C03579=1018.745,297.006,-138.306,170.005,50.463,159.764
C03580=1018.752,297.252,-138.337,170.011,50.459,159.764
C03581=1018.758,297.501,-138.369,170.016,50.455,159.763
C03582=1018.764,297.748,-138.401,170.022,50.451,159.763
C03583=1018.770,297.997,-138.433,170.026,50.447,159.763
C03584=1018.777,298.245,-138.464,170.033,50.443,159.764
C03585=1018.783,298.492,-138.497,170.038,50.439,159.764
C03586=1018.789,298.740,-138.529,170.043,50.435,159.764
C03587=1018.795,298.988,-138.560,170.048,50.431,159.763
C03588=1018.801,299.236,-138.592,170.055,50.427,159.764
C03589=1018.808,299.483,-138.624,170.059,50.423,159.764
C03590=1018.814,299.731,-138.656,170.065,50.418,159.764
C03591=1018.821,299.979,-138.688,170.071,50.414,159.764
C03592=1018.827,300.227,-138.720,170.076,50.411,159.764
C03593=1018.833,300.475,-138.753,170.082,50.406,159.764
C03594=1018.840,300.723,-138.784,170.087,50.402,159.764
C03595=1018.846,300.970,-138.817,170.094,50.399,159.764
C03596=1018.853,301.218,-138.848,170.098,50.395,159.764
C03597=1018.859,301.467,-138.880,170.104,50.390,159.764
C03598=1018.866,301.714,-138.912,170.110,50.387,159.764
C03599=1018.872,301.962,-138.944,170.115,50.383,159.764
C03600=1018.879,302.210,-138.977,170.121,50.379,159.764
C03601=1018.885,302.458,-139.009,170.127,50.375,159.764
C03602=1018.892,302.705,-139.041,170.132,50.371,159.764
C03603=1018.898,302.953,-139.073,170.138,50.367,159.764
C03604=1018.905,303.201,-139.105,170.144,50.363,159.764
C03605=1018.911,303.449,-139.137,170.149,50.360,159.764
C03606=1018.918,303.696,-139.170,170.155,50.355,159.764
C03607=1018.924,303.944,-139.202,170.160,50.352,159.764
C03608=1018.931,304.192,-139.234,170.166,50.348,159.764
C03609=1018.937,304.440,-139.266,170.171,50.344,159.764
C03610=1018.944,304.687,-139.298,170.177,50.341,159.765
C03611=1018.950,304.935,-139.331,170.183,50.336,159.765
C03612=1018.957,305.183,-139.363,170.189,50.333,159.765
C03613=1018.964,305.431,-139.395,170.194,50.328,159.765
C03614=1018.970,305.679,-139.428,170.200,50.325,159.765
C03615=1018.977,305.926,-139.459,170.206,50.321,159.765
C03616=1018.983,306.174,-139.492,170.212,50.317,159.765
C03617=1018.990,306.421,-139.524,170.217,50.314,159.765
C03618=1018.997,306.670,-139.557,170.223,50.309,159.765
C03619=1019.003,306.917,-139.589,170.228,50.306,159.765
C03620=1019.010,307.163,-139.621,170.235,50.302,159.765
C03621=1019.016,307.409,-139.653,170.240,50.299,159.766
C03622=1019.023,307.655,-139.686,170.246,50.295,159.765
C03623=1019.030,307.901,-139.718,170.251,50.291,159.766
C03624=1019.036,308.146,-139.751,170.257,50.288,159.766
C03625=1019.043,308.391,-139.783,170.263,50.284,159.766
C03626=1019.050,308.637,-139.815,170.268,50.280,159.766
C03627=1019.057,308.884,-139.847,170.275,50.276,159.766
C03628=1019.063,309.131,-139.880,170.280,50.273,159.766
C03629=1019.070,309.379,-139.912,170.286,50.269,159.766
C03630=1019.076,309.626,-139.944,170.292,50.266,159.767
C03631=1019.083,309.874,-139.977,170.297,50.262,159.767
C03632=1019.090,310.122,-140.011,170.304,50.258,159.767
C03633=1019.096,310.369,-140.044,170.309,50.255,159.767
C03634=1019.102,310.617,-140.076,170.315,50.252,159.767
C03635=1019.109,310.864,-140.110,170.321,50.248,159.767
C03636=1019.115,311.112,-140.144,170.327,50.245,159.768
C03637=1019.121,311.360,-140.176,170.332,50.241,159.768
C03638=1019.128,311.607,-140.210,170.339,50.238,159.768
C03639=1019.135,311.855,-140.243,170.344,50.234,159.768
C03640=1019.141,312.103,-140.276,170.350,50.231,159.768
C03641=1019.147,312.350,-140.310,170.356,50.228,159.768
C03642=1019.154,312.598,-140.343,170.362,50.224,159.769
C03643=1019.161,312.845,-140.376,170.367,50.221,159.769
C03644=1019.167,313.093,-140.409,170.374,50.217,159.769
C03645=1019.173,313.342,-140.443,170.379,50.215,159.769
C03646=1019.180,313.589,-140.476,170.385,50.211,159.769
C03647=1019.186,313.837,-140.509,170.391,50.208,159.770
C03648=1019.193,314.084,-140.543,170.397,50.204,159.770
C03649=1019.200,314.331,-140.576,170.404,50.201,159.770
C03650=1019.206,314.579,-140.610,170.409,50.197,159.770
C03651=1019.212,314.826,-140.643,170.415,50.194,159.770
C03652=1019.219,315.075,-140.677,170.421,50.191,159.771
C03653=1019.226,315.322,-140.710,170.427,50.187,159.771
C03654=1019.232,315.570,-140.744,170.433,50.185,159.771
C03655=1019.239,315.817,-140.777,170.439,50.181,159.771
C03656=1019.246,316.065,-140.811,170.444,50.178,159.772
C03657=1019.252,316.312,-140.844,170.451,50.175,159.772
C03658=1019.259,316.560,-140.878,170.457,50.171,159.772
C03659=1019.265,316.807,-140.912,170.463,50.168,159.772
C03660=1019.272,317.056,-140.945,170.469,50.165,159.773
C03661=1019.279,317.303,-140.979,170.475,50.162,159.773
C03662=1019.285,317.551,-141.013,170.481,50.158,159.773
C03663=1019.292,317.798,-141.046,170.487,50.156,159.773
C03664=1019.299,318.046,-141.079,170.493,50.152,159.774
C03665=1019.306,318.294,-141.113,170.500,50.149,159.774
C03666=1019.312,318.542,-141.147,170.505,50.146,159.774
C03667=1019.319,318.789,-141.181,170.512,50.143,159.775
C03668=1019.326,319.036,-141.215,170.518,50.139,159.775
C03669=1019.333,319.284,-141.248,170.523,50.136,159.775
C03670=1019.339,319.531,-141.283,170.530,50.133,159.775
C03671=1019.346,319.779,-141.316,170.535,50.130,159.776
C03672=1019.353,320.027,-141.349,170.542,50.127,159.776
C03673=1019.360,320.274,-141.383,170.549,50.124,159.776
C03674=1019.366,320.522,-141.417,170.554,50.121,159.776
C03675=1019.374,320.770,-141.451,170.561,50.118,159.777
C03676=1019.381,321.017,-141.485,170.566,50.115,159.777
C03677=1019.387,321.264,-141.518,170.572,50.111,159.777
C03678=1019.394,321.512,-141.553,170.579,50.108,159.778
C03679=1019.401,321.760,-141.587,170.585,50.106,159.778
C03680=1019.408,322.009,-141.621,170.591,50.103,159.778
C03681=1019.415,322.258,-141.656,170.598,50.099,159.779
C03682=1019.422,322.507,-141.689,170.603,50.096,159.779
C03683=1019.429,322.756,-141.724,170.610,50.093,159.779
C03684=1019.437,323.004,-141.758,170.617,50.090,159.780
C03685=1019.443,323.252,-141.792,170.622,50.088,159.780
C03686=1019.450,323.498,-141.826,170.629,50.084,159.780
C03687=1019.457,323.746,-141.859,170.635,50.081,159.781
C03688=1019.463,323.994,-141.894,170.642,50.078,159.781
C03689=1019.471,324.241,-141.928,170.647,50.075,159.781
C03690=1019.478,324.489,-141.962,170.654,50.072,159.782
C03691=1019.485,324.737,-141.996,170.661,50.069,159.782
C03692=1019.492,324.985,-142.030,170.666,50.066,159.782
C03693=1019.499,325.232,-142.065,170.673,50.063,159.783
C03694=1019.506,325.479,-142.099,170.680,50.060,159.783
C03695=1019.514,325.727,-142.133,170.685,50.058,159.783
C03696=1019.520,325.974,-142.168,170.692,50.055,159.784
C03697=1019.528,326.222,-142.202,170.699,50.052,159.784
C03698=1019.535,326.469,-142.236,170.704,50.049,159.784
C03699=1019.542,326.717,-142.270,170.711,50.046,159.785
C03700=1019.548,326.964,-142.306,170.718,50.043,159.785
C03701=1019.555,327.212,-142.339,170.724,50.041,159.786
C03702=1019.562,327.459,-142.375,170.730,50.038,159.786
C03703=1019.569,327.707,-142.410,170.737,50.035,159.787
C03704=1019.576,327.954,-142.444,170.743,50.032,159.787
C03705=1019.583,328.202,-142.479,170.750,50.030,159.787
C03706=1019.590,328.449,-142.514,170.756,50.027,159.788
C03707=1019.597,328.697,-142.549,170.762,50.024,159.788
C03708=1019.604,328.944,-142.583,170.769,50.022,159.789
C03709=1019.610,329.192,-142.618,170.776,50.019,159.789
C03710=1019.617,329.439,-142.653,170.781,50.016,159.789
C03711=1019.625,329.686,-142.688,170.788,50.014,159.790
C03712=1019.632,329.933,-142.723,170.795,50.011,159.790
C03713=1019.639,330.182,-142.758,170.801,50.009,159.791
C03714=1019.645,330.429,-142.793,170.808,50.006,159.791
C03715=1019.653,330.676,-142.827,170.814,50.003,159.792
C03716=1019.660,330.924,-142.862,170.821,50.000,159.792
C03717=1019.666,331.171,-142.897,170.827,49.998,159.793
C03718=1019.673,331.419,-142.933,170.834,49.995,159.793
C03719=1019.681,331.666,-142.967,170.841,49.992,159.793
C03720=1019.688,331.914,-143.003,170.847,49.990,159.794
C03721=1019.695,332.161,-143.038,170.853,49.987,159.794
C03722=1019.702,332.408,-143.072,170.860,49.985,159.795
C03723=1019.710,332.656,-143.108,170.867,49.983,159.796
C03724=1019.716,332.904,-143.143,170.873,49.980,159.796
C03725=1019.723,333.151,-143.178,170.880,49.978,159.796
C03726=1019.730,333.398,-143.214,170.887,49.975,159.797
C03727=1019.738,333.646,-143.249,170.893,49.972,159.797
C03728=1019.744,333.893,-143.285,170.900,49.970,159.798
C03729=1019.751,334.140,-143.320,170.907,49.968,159.798
C03730=1019.758,334.387,-143.356,170.914,49.965,159.799
C03731=1019.766,334.635,-143.391,170.919,49.963,159.799
C03732=1019.772,334.883,-143.426,170.926,49.960,159.800
C03733=1019.779,335.129,-143.462,170.933,49.958,159.801
C03734=1019.787,335.377,-143.498,170.939,49.956,159.801
C03735=1019.794,335.625,-143.533,170.946,49.954,159.802
C03736=1019.801,335.872,-143.569,170.953,49.951,159.802
C03737=1019.808,336.120,-143.604,170.960,49.948,159.803
C03738=1019.815,336.366,-143.640,170.966,49.946,159.803
C03739=1019.823,336.614,-143.675,170.973,49.944,159.804
C03740=1019.830,336.860,-143.710,170.980,49.941,159.804
C03741=1019.837,337.106,-143.747,170.987,49.939,159.805
C03742=1019.844,337.352,-143.782,170.993,49.937,159.805
C03743=1019.851,337.599,-143.818,171.000,49.935,159.806
C03744=1019.859,337.844,-143.852,171.007,49.932,159.806
C03745=1019.866,338.091,-143.888,171.014,49.930,159.807
C03746=1019.873,338.336,-143.924,171.020,49.928,159.808
C03747=1019.880,338.583,-143.960,171.027,49.926,159.808
C03748=1019.887,338.830,-143.996,171.034,49.923,159.809
C03749=1019.895,339.078,-144.031,171.042,49.921,159.810
C03750=1019.902,339.324,-144.067,171.049,49.919,159.810
C03751=1019.909,339.572,-144.103,171.055,49.917,159.811
C03752=1019.917,339.819,-144.139,171.062,49.915,159.811
C03753=1019.924,340.066,-144.176,171.069,49.912,159.812
C03754=1019.931,340.315,-144.211,171.076,49.911,159.813
C03755=1019.938,340.561,-144.247,171.083,49.908,159.813
C03756=1019.946,340.809,-144.283,171.089,49.906,159.814
C03757=1019.952,341.056,-144.320,171.096,49.904,159.814
C03758=1019.960,341.303,-144.356,171.104,49.902,159.815
C03759=1019.967,341.551,-144.392,171.111,49.900,159.816
C03760=1019.974,341.797,-144.428,171.118,49.897,159.816
C03761=1019.981,342.045,-144.465,171.124,49.896,159.817
C03762=1019.989,342.293,-144.501,171.131,49.894,159.817
C03763=1019.996,342.539,-144.537,171.139,49.892,159.818
C03764=1020.004,342.786,-144.574,171.146,49.889,159.819
C03765=1020.011,343.034,-144.611,171.153,49.888,159.820
C03766=1020.018,343.281,-144.647,171.160,49.885,159.820
C03767=1020.026,343.528,-144.683,171.166,49.884,159.821
C03768=1020.033,343.776,-144.720,171.173,49.882,159.821
C03769=1020.040,344.023,-144.756,171.181,49.880,159.822
C03770=1020.048,344.269,-144.792,171.188,49.877,159.823
C03771=1020.055,344.517,-144.829,171.195,49.876,159.824
C03772=1020.062,344.765,-144.865,171.202,49.873,159.824
C03773=1020.070,345.011,-144.902,171.210,49.872,159.825
C03774=1020.077,345.259,-144.939,171.217,49.870,159.826
C03775=1020.085,345.507,-144.975,171.223,49.868,159.826
C03776=1020.092,345.753,-145.012,171.230,49.866,159.827
C03777=1020.099,346.001,-145.049,171.238,49.864,159.828
C03778=1020.107,346.247,-145.086,171.245,49.862,159.828
C03779=1020.115,346.495,-145.122,171.252,49.860,159.829
C03780=1020.122,346.742,-145.159,171.260,49.859,159.830
C03781=1020.130,346.989,-145.196,171.267,49.857,159.831
C03782=1020.138,347.236,-145.233,171.274,49.854,159.831
C03783=1020.145,347.484,-145.269,171.281,49.853,159.832
C03784=1020.152,347.731,-145.307,171.289,49.851,159.833
C03785=1020.160,347.978,-145.344,171.296,49.849,159.834
C03786=1020.167,348.226,-145.381,171.304,49.848,159.834
C03787=1020.175,348.473,-145.418,171.310,49.846,159.835
C03788=1020.182,348.720,-145.455,171.317,49.844,159.836
C03789=1020.190,348.966,-145.492,171.325,49.843,159.837
C03790=1020.197,349.214,-145.529,171.332,49.841,159.837
C03791=1020.205,349.461,-145.566,171.340,49.839,159.838
C03792=1020.212,349.708,-145.603,171.347,49.837,159.839
C03793=1020.220,349.955,-145.641,171.354,49.836,159.840
C03794=1020.228,350.202,-145.678,171.362,49.834,159.841
C03795=1020.235,350.449,-145.715,171.369,49.832,159.841
C03796=1020.242,350.696,-145.753,171.376,49.830,159.842
C03797=1020.250,350.943,-145.790,171.384,49.829,159.843
C03798=1020.257,351.190,-145.827,171.392,49.828,159.844
C03799=1020.265,351.437,-145.864,171.399,49.826,159.845
C03800=1020.272,351.682,-145.901,171.406,49.824,159.845
C03801=1020.280,351.927,-145.938,171.414,49.822,159.846
C03802=1020.288,352.171,-145.975,171.421,49.821,159.847
C03803=1020.295,352.416,-146.012,171.429,49.820,159.848
C03804=1020.302,352.661,-146.049,171.436,49.818,159.849
C03805=1020.310,352.905,-146.086,171.444,49.816,159.850
C03806=1020.318,353.150,-146.124,171.451,49.814,159.850
C03807=1020.326,353.394,-146.161,171.459,49.813,159.851
C03808=1020.334,353.641,-146.198,171.466,49.811,159.852
C03809=1020.341,353.888,-146.236,171.474,49.810,159.853
C03810=1020.350,354.135,-146.274,171.481,49.809,159.854
C03811=1020.357,354.382,-146.311,171.489,49.807,159.855
C03812=1020.364,354.629,-146.349,171.497,49.806,159.856
C03813=1020.372,354.876,-146.387,171.504,49.804,159.856
C03814=1020.380,355.124,-146.425,171.512,49.803,159.857
C03815=1020.388,355.370,-146.463,171.519,49.801,159.858
C03816=1020.395,355.617,-146.500,171.527,49.800,159.859
C03817=1020.403,355.864,-146.539,171.535,49.799,159.860
C03818=1020.410,356.111,-146.576,171.542,49.797,159.861
C03819=1020.418,356.358,-146.614,171.550,49.796,159.862
C03820=1020.427,356.605,-146.652,171.557,49.794,159.863
C03821=1020.434,356.852,-146.690,171.566,49.793,159.864
C03822=1020.442,357.099,-146.729,171.574,49.792,159.865
C03823=1020.450,357.346,-146.766,171.582,49.791,159.866
C03824=1020.458,357.594,-146.805,171.589,49.789,159.866
C03825=1020.465,357.840,-146.843,171.597,49.788,159.867
C03826=1020.474,358.087,-146.881,171.604,49.787,159.868
C03827=1020.481,358.334,-146.919,171.612,49.785,159.869
C03828=1020.490,358.581,-146.957,171.620,49.784,159.870
C03829=1020.497,358.828,-146.995,171.628,49.782,159.871
C03830=1020.505,359.075,-147.034,171.636,49.781,159.872
C03831=1020.513,359.322,-147.072,171.644,49.780,159.873
C03832=1020.521,359.569,-147.111,171.652,49.779,159.874
C03833=1020.529,359.815,-147.149,171.659,49.778,159.875
C03834=1020.537,360.063,-147.188,171.667,49.777,159.876
C03835=1020.544,360.309,-147.226,171.676,49.775,159.877
C03836=1020.552,360.556,-147.265,171.684,49.774,159.878
C03837=1020.561,360.803,-147.303,171.691,49.773,159.879
C03838=1020.568,361.050,-147.341,171.699,49.772,159.880
C03839=1020.575,361.298,-147.381,171.707,49.771,159.881
C03840=1020.583,361.543,-147.420,171.716,49.770,159.882
C03841=1020.591,361.791,-147.458,171.724,49.769,159.883
C03842=1020.600,362.038,-147.497,171.732,49.768,159.884
C03843=1020.607,362.284,-147.535,171.739,49.766,159.885
C03844=1020.616,362.531,-147.574,171.747,49.765,159.886
C03845=1020.624,362.778,-147.613,171.756,49.764,159.888
C03846=1020.631,363.025,-147.651,171.764,49.763,159.889
C03847=1020.639,363.272,-147.691,171.772,49.762,159.890
C03848=1020.647,363.519,-147.730,171.780,49.762,159.891
C03849=1020.656,363.765,-147.769,171.789,49.760,159.892
C03850=1020.664,364.013,-147.808,171.796,49.759,159.893
C03851=1020.672,364.258,-147.847,171.805,49.759,159.894
C03852=1020.680,364.506,-147.885,171.813,49.757,159.895
C03853=1020.688,364.752,-147.925,171.821,49.757,159.896
C03854=1020.696,365.000,-147.964,171.829,49.755,159.897
C03855=1020.704,365.246,-148.003,171.837,49.754,159.898
C03856=1020.713,365.493,-148.042,171.846,49.753,159.899
C03857=1020.721,365.740,-148.081,171.854,49.752,159.900
C03858=1020.729,365.986,-148.120,171.862,49.752,159.902
C03859=1020.737,366.233,-148.159,171.871,49.751,159.903
C03860=1020.745,366.482,-148.199,171.879,49.750,159.904
C03861=1020.753,366.732,-148.238,171.888,49.749,159.905
C03862=1020.762,366.981,-148.278,171.896,49.748,159.906
C03863=1020.770,367.231,-148.318,171.905,49.747,159.907
C03864=1020.779,367.478,-148.357,171.913,49.746,159.908
C03865=1020.787,367.725,-148.397,171.921,49.746,159.910
C03866=1020.796,367.971,-148.436,171.930,49.744,159.911
C03867=1020.804,368.218,-148.476,171.938,49.744,159.912
C03868=1020.812,368.465,-148.515,171.947,49.743,159.913
C03869=1020.820,368.712,-148.555,171.955,49.742,159.914
C03870=1020.828,368.958,-148.594,171.963,49.742,159.916
C03871=1020.836,369.205,-148.634,171.973,49.741,159.917
C03872=1020.845,369.451,-148.674,171.981,49.741,159.918
C03873=1020.852,369.698,-148.714,171.990,49.740,159.919
C03874=1020.861,369.945,-148.754,171.998,49.739,159.920
C03875=1020.869,370.192,-148.793,172.007,49.738,159.922
C03876=1020.877,370.437,-148.833,172.015,49.738,159.923
C03877=1020.885,370.684,-148.873,172.023,49.737,159.924
C03878=1020.894,370.932,-148.913,172.033,49.736,159.925
C03879=1020.902,371.178,-148.954,172.041,49.736,159.927
C03880=1020.911,371.425,-148.993,172.050,49.735,159.928
C03881=1020.919,371.671,-149.034,172.058,49.734,159.929
C03882=1020.927,371.917,-149.073,172.067,49.734,159.930
C03883=1020.936,372.165,-149.113,172.076,49.734,159.932
C03884=1020.944,372.411,-149.153,172.085,49.733,159.933
C03885=1020.953,372.657,-149.193,172.093,49.732,159.934
C03886=1020.961,372.905,-149.234,172.102,49.732,159.936
C03887=1020.970,373.151,-149.274,172.111,49.731,159.937
C03888=1020.978,373.397,-149.314,172.120,49.731,159.938
C03889=1020.987,373.644,-149.354,172.129,49.730,159.939
C03890=1020.995,373.890,-149.395,172.137,49.730,159.941
C03891=1021.004,374.137,-149.434,172.146,49.729,159.942
C03892=1021.012,374.384,-149.475,172.155,49.729,159.943
C03893=1021.021,374.630,-149.515,172.164,49.728,159.945
C03894=1021.030,374.877,-149.556,172.173,49.728,159.946
C03895=1021.038,375.123,-149.596,172.182,49.727,159.947
C03896=1021.047,375.371,-149.636,172.191,49.727,159.949
C03897=1021.055,375.617,-149.676,172.200,49.726,159.950
C03898=1021.064,375.864,-149.717,172.209,49.726,159.951
C03899=1021.073,376.110,-149.757,172.218,49.725,159.953
C03900=1021.081,376.357,-149.798,172.227,49.725,159.954
C03901=1021.089,376.603,-149.839,172.236,49.725,159.955
C03902=1021.098,376.850,-149.880,172.245,49.725,159.957
C03903=1021.107,377.095,-149.921,172.254,49.724,159.958
C03904=1021.116,377.342,-149.962,172.263,49.724,159.960
C03905=1021.124,377.588,-150.002,172.272,49.724,159.961
C03906=1021.132,377.835,-150.043,172.282,49.723,159.962
C03907=1021.141,378.081,-150.085,172.290,49.723,159.964
C03908=1021.150,378.328,-150.125,172.300,49.723,159.965
C03909=1021.159,378.575,-150.166,172.309,49.723,159.967
C03910=1021.167,378.820,-150.208,172.319,49.723,159.968
C03911=1021.176,379.067,-150.249,172.327,49.723,159.970
C03912=1021.185,379.314,-150.290,172.337,49.722,159.971
C03913=1021.193,379.560,-150.331,172.346,49.722,159.973
C03914=1021.202,379.806,-150.372,172.356,49.722,159.974
C03915=1021.211,380.053,-150.413,172.364,49.722,159.975
C03916=1021.219,380.299,-150.454,172.374,49.722,159.977
C03917=1021.228,380.545,-150.496,172.383,49.721,159.978
C03918=1021.237,380.792,-150.537,172.393,49.721,159.980
C03919=1021.246,381.038,-150.579,172.403,49.721,159.982
C03920=1021.256,381.310,-150.624,172.412,49.721,159.983
C03921=1021.265,381.581,-150.669,172.423,49.721,159.985
C03922=1021.276,381.852,-150.715,172.434,49.721,159.986
C03923=1021.285,382.124,-150.761,172.444,49.721,159.988
C03924=1021.294,382.370,-150.803,172.453,49.721,159.990
C03925=1021.303,382.617,-150.844,172.463,49.721,159.991
C03926=1021.313,382.863,-150.885,172.473,49.721,159.993
C03927=1021.322,383.109,-150.927,172.482,49.721,159.994
C03928=1021.331,383.356,-150.969,172.492,49.720,159.996
C03929=1021.339,383.602,-151.010,172.502,49.721,159.997
C03930=1021.348,383.848,-151.052,172.511,49.720,159.999
C03931=1021.357,384.095,-151.094,172.521,49.721,160.001
C03932=1021.367,384.341,-151.135,172.531,49.721,160.002
C03933=1021.376,384.587,-151.177,172.540,49.721,160.004
C03934=1021.385,384.833,-151.218,172.550,49.721,160.005
C03935=1021.394,385.080,-151.260,172.560,49.721,160.007
C03936=1021.403,385.326,-151.302,172.570,49.721,160.008
C03937=1021.412,385.573,-151.344,172.580,49.721,160.010
C03938=1021.421,385.819,-151.386,172.589,49.721,160.012
C03939=1021.430,386.065,-151.428,172.599,49.721,160.013
C03940=1021.440,386.311,-151.471,172.609,49.721,160.015
C03941=1021.449,386.558,-151.512,172.619,49.722,160.017
C03942=1021.458,386.803,-151.555,172.629,49.722,160.018
C03943=1021.467,387.050,-151.597,172.638,49.722,160.020
C03944=1021.477,387.296,-151.639,172.648,49.723,160.022
C03945=1021.486,387.542,-151.681,172.658,49.723,160.023
C03946=1021.495,387.788,-151.723,172.669,49.723,160.025
C03947=1021.505,388.035,-151.766,172.679,49.723,160.027
C03948=1021.513,388.281,-151.808,172.689,49.723,160.028
C03949=1021.522,388.527,-151.851,172.699,49.724,160.030
C03950=1021.531,388.773,-151.893,172.709,49.724,160.032
C03951=1021.541,389.019,-151.936,172.719,49.725,160.034
C03952=1021.550,389.265,-151.979,172.729,49.725,160.035
C03953=1021.559,389.512,-152.022,172.740,49.725,160.037
C03954=1021.569,389.757,-152.064,172.749,49.725,160.039
C03955=1021.578,390.003,-152.107,172.760,49.726,160.041
C03956=1021.588,390.250,-152.150,172.770,49.726,160.042
C03957=1021.596,390.496,-152.193,172.781,49.727,160.044
C03958=1021.606,390.742,-152.235,172.791,49.727,160.046
C03959=1021.615,390.988,-152.278,172.801,49.727,160.048
C03960=1021.625,391.234,-152.321,172.811,49.728,160.050
C03961=1021.634,391.480,-152.363,172.822,49.728,160.051
C03962=1021.644,391.727,-152.407,172.832,49.729,160.053
C03963=1021.653,391.972,-152.450,172.842,49.730,160.055
C03964=1021.663,392.218,-152.492,172.853,49.730,160.057
C03965=1021.671,392.464,-152.536,172.863,49.731,160.059
C03966=1021.682,392.710,-152.579,172.873,49.731,160.060
C03967=1021.691,392.957,-152.622,172.884,49.732,160.062
C03968=1021.700,393.202,-152.666,172.895,49.732,160.064
C03969=1021.710,393.449,-152.708,172.905,49.733,160.066
C03970=1021.720,393.694,-152.752,172.916,49.734,160.068
C03971=1021.729,393.940,-152.795,172.926,49.734,160.070
C03972=1021.739,394.186,-152.838,172.937,49.734,160.072
C03973=1021.748,394.432,-152.883,172.948,49.735,160.074
C03974=1021.758,394.679,-152.925,172.958,49.736,160.076
C03975=1021.767,394.924,-152.969,172.969,49.737,160.078
C03976=1021.777,395.170,-153.013,172.979,49.737,160.079
C03977=1021.787,395.416,-153.056,172.990,49.738,160.081
C03978=1021.796,395.663,-153.099,173.001,49.739,160.083
C03979=1021.806,395.909,-153.143,173.012,49.739,160.085
C03980=1021.819,396.217,-153.198,173.026,49.740,160.088
C03981=1021.831,396.525,-153.253,173.039,49.742,160.090
C03982=1021.843,396.834,-153.307,173.053,49.743,160.093
C03983=1021.855,397.142,-153.363,173.067,49.744,160.095
C03984=1021.865,397.388,-153.407,173.078,49.744,160.097
C03985=1021.875,397.634,-153.450,173.088,49.745,160.099
C03986=1021.884,397.880,-153.494,173.100,49.746,160.101
C03987=1021.895,398.126,-153.539,173.110,49.747,160.103
C03988=1021.904,398.372,-153.583,173.122,49.748,160.105
C03989=1021.914,398.618,-153.627,173.133,49.748,160.107
C03990=1021.924,398.863,-153.671,173.144,49.750,160.110
C03991=1021.934,399.109,-153.715,173.155,49.750,160.111
C03992=1021.944,399.355,-153.759,173.167,49.751,160.114
C03993=1021.954,399.601,-153.804,173.177,49.752,160.116
C03994=1021.964,399.847,-153.849,173.189,49.753,160.118
C03995=1021.974,400.093,-153.892,173.200,49.754,160.120
C03996=1021.984,400.338,-153.937,173.212,49.755,160.122
C03997=1021.993,400.584,-153.981,173.222,49.756,160.124
C03998=1022.004,400.830,-154.026,173.234,49.757,160.126
C03999=1022.014,401.076,-154.071,173.245,49.758,160.128
C04000=1022.024,401.321,-154.115,173.257,49.759,160.131
C04001=1022.033,401.567,-154.160,173.269,49.760,160.133
C04002=1022.043,401.814,-154.205,173.279,49.762,160.135
C04003=1022.053,402.059,-154.249,173.291,49.763,160.137
C04004=1022.063,402.304,-154.294,173.302,49.764,160.139
C04005=1022.074,402.550,-154.339,173.314,49.765,160.141
C04006=1022.084,402.795,-154.384,173.326,49.766,160.144
C04007=1022.093,403.041,-154.429,173.338,49.767,160.146
C04008=1022.104,403.287,-154.474,173.349,49.768,160.148
C04009=1022.114,403.532,-154.519,173.361,49.769,160.150
C04010=1022.125,403.778,-154.564,173.373,49.770,160.152
C04011=1022.134,404.024,-154.609,173.385,49.772,160.155
C04012=1022.145,404.270,-154.655,173.396,49.773,160.157
C04013=1022.155,404.515,-154.699,173.408,49.774,160.159
C04014=1022.165,404.761,-154.745,173.420,49.776,160.162
C04015=1022.176,405.006,-154.790,173.431,49.777,160.164
C04016=1022.186,405.252,-154.835,173.443,49.778,160.166
C04017=1022.196,405.497,-154.880,173.455,49.779,160.168
C04018=1022.206,405.743,-154.925,173.467,49.781,160.171
C04019=1022.217,405.989,-154.971,173.479,49.782,160.173
C04020=1022.227,406.235,-155.017,173.491,49.783,160.175
C04021=1022.237,406.480,-155.062,173.503,49.785,160.178
C04022=1022.249,406.725,-155.107,173.516,49.786,160.180
C04023=1022.259,406.971,-155.153,173.527,49.787,160.182
C04024=1022.270,407.217,-155.199,173.539,49.789,160.185
C04025=1022.280,407.462,-155.244,173.551,49.790,160.187
C04026=1022.290,407.708,-155.290,173.563,49.792,160.190
C04027=1022.301,407.954,-155.335,173.576,49.793,160.192
C04028=1022.312,408.199,-155.380,173.588,49.795,160.194
C04029=1022.323,408.445,-155.426,173.600,49.796,160.197
C04030=1022.333,408.690,-155.472,173.613,49.798,160.199
C04031=1022.344,408.936,-155.518,173.625,49.799,160.202
C04032=1022.354,409.181,-155.564,173.637,49.801,160.204
C04033=1022.365,409.427,-155.610,173.650,49.802,160.207
C04034=1022.376,409.672,-155.657,173.662,49.803,160.209
C04035=1022.387,409.918,-155.703,173.675,49.806,160.212
C04036=1022.397,410.163,-155.748,173.688,49.807,160.214
C04037=1022.407,410.408,-155.796,173.700,49.808,160.216
C04038=1022.418,410.654,-155.842,173.712,49.811,160.219
C04039=1022.429,410.899,-155.888,173.725,49.812,160.222
C04040=1022.444,411.231,-155.951,173.743,49.814,160.225
C04041=1022.458,411.561,-156.013,173.760,49.816,160.228
C04042=1022.473,411.893,-156.076,173.776,49.819,160.232
C04043=1022.488,412.224,-156.139,173.794,49.821,160.235
C04044=1022.498,412.470,-156.186,173.807,49.823,160.238
C04045=1022.509,412.715,-156.232,173.819,49.825,160.241
C04046=1022.520,412.960,-156.279,173.833,49.826,160.243
C04047=1022.531,413.206,-156.326,173.846,49.828,160.246
C04048=1022.542,413.451,-156.372,173.858,49.830,160.248
C04049=1022.554,413.697,-156.419,173.871,49.831,160.251
C04050=1022.564,413.942,-156.467,173.885,49.833,160.254
C04051=1022.575,414.187,-156.513,173.897,49.835,160.256
C04052=1022.587,414.433,-156.560,173.911,49.837,160.259
C04053=1022.598,414.678,-156.607,173.924,49.839,160.262
C04054=1022.609,414.923,-156.654,173.937,49.840,160.264
C04055=1022.621,415.169,-156.701,173.950,49.842,160.267
C04056=1022.631,415.414,-156.748,173.964,49.845,160.270
C04057=1022.643,415.659,-156.796,173.977,49.847,160.273
C04058=1022.653,415.905,-156.843,173.990,49.848,160.275
C04059=1022.665,416.150,-156.891,174.004,49.851,160.278
C04060=1022.676,416.395,-156.938,174.017,49.852,160.281
C04061=1022.687,416.640,-156.986,174.031,49.855,160.284
C04062=1022.698,416.886,-157.033,174.044,49.857,160.286
C04063=1022.709,417.131,-157.081,174.057,49.859,160.289
C04064=1022.721,417.375,-157.128,174.071,49.861,160.292
C04065=1022.731,417.621,-157.176,174.085,49.863,160.295
C04066=1022.743,417.866,-157.224,174.098,49.865,160.298
C04067=1022.755,418.111,-157.271,174.112,49.867,160.301
C04068=1022.766,418.357,-157.320,174.126,49.869,160.304
C04069=1022.778,418.602,-157.367,174.140,49.871,160.306
C04070=1022.788,418.847,-157.415,174.154,49.873,160.309
C04071=1022.800,419.092,-157.463,174.168,49.875,160.312
C04072=1022.811,419.337,-157.511,174.182,49.878,160.315
C04073=1022.823,419.582,-157.559,174.195,49.880,160.318
C04074=1022.835,419.827,-157.607,174.209,49.882,160.321
C04075=1022.846,420.072,-157.655,174.224,49.884,160.324
C04076=1022.858,420.317,-157.703,174.238,49.886,160.327
C04077=1022.870,420.563,-157.752,174.251,49.888,160.330
C04078=1022.882,420.808,-157.800,174.265,49.891,160.333
C04079=1022.894,421.053,-157.847,174.280,49.893,160.336
C04080=1022.905,421.298,-157.896,174.294,49.895,160.339
C04081=1022.917,421.543,-157.944,174.308,49.898,160.342
C04082=1022.929,421.789,-157.993,174.323,49.900,160.345
C04083=1022.940,422.034,-158.042,174.337,49.902,160.348
C04084=1022.952,422.278,-158.090,174.352,49.905,160.351
C04085=1022.964,422.523,-158.139,174.366,49.907,160.354
C04086=1022.975,422.769,-158.188,174.380,49.910,160.357
C04087=1022.987,423.013,-158.236,174.395,49.912,160.360
C04088=1022.999,423.258,-158.285,174.409,49.915,160.364
C04089=1023.011,423.503,-158.335,174.424,49.917,160.367
C04090=1023.023,423.748,-158.383,174.439,49.919,160.370
C04091=1023.034,423.993,-158.432,174.453,49.922,160.373
C04092=1023.047,424.238,-158.481,174.469,49.924,160.376
C04093=1023.059,424.483,-158.530,174.483,49.927,160.379
C04094=1023.071,424.728,-158.579,174.498,49.929,160.382
C04095=1023.083,424.972,-158.628,174.513,49.932,160.386
C04096=1023.095,425.217,-158.678,174.528,49.935,160.389
C04097=1023.107,425.463,-158.727,174.543,49.937,160.392
C04098=1023.120,425.708,-158.776,174.558,49.940,160.395
C04099=1023.131,425.952,-158.826,174.573,49.942,160.399
C04100=1023.145,426.222,-158.880,174.590,49.945,160.402
C04101=1023.158,426.491,-158.935,174.607,49.948,160.406
C04102=1023.171,426.761,-158.990,174.623,49.951,160.410
C04103=1023.185,427.031,-159.044,174.640,49.954,160.413
C04104=1023.197,427.275,-159.094,174.655,49.957,160.417
C04105=1023.209,427.520,-159.144,174.670,49.960,160.420
C04106=1023.221,427.764,-159.194,174.686,49.963,160.423
C04107=1023.234,428.009,-159.244,174.701,49.965,160.427
C04108=1023.246,428.254,-159.294,174.717,49.968,160.430
C04109=1023.258,428.499,-159.344,174.732,49.971,160.434
C04110=1023.271,428.744,-159.395,174.749,49.974,160.437
C04111=1023.284,428.988,-159.444,174.764,49.977,160.441
C04112=1023.296,429.233,-159.494,174.780,49.979,160.444
C04113=1023.308,429.478,-159.544,174.796,49.982,160.447
C04114=1023.321,429.722,-159.595,174.811,49.985,160.451
C04115=1023.333,429.967,-159.645,174.827,49.988,160.454
C04116=1023.346,430.212,-159.695,174.843,49.990,160.458
C04117=1023.358,430.456,-159.746,174.859,49.994,160.461
C04118=1023.371,430.700,-159.796,174.875,49.997,160.465
C04119=1023.384,430.945,-159.846,174.892,50.000,160.469
C04120=1023.397,431.190,-159.897,174.907,50.003,160.472
C04121=1023.409,431.434,-159.948,174.924,50.006,160.476
C04122=1023.422,431.678,-159.998,174.940,50.008,160.479
C04123=1023.434,431.923,-160.049,174.956,50.012,160.483
C04124=1023.448,432.168,-160.099,174.973,50.015,160.487
C04125=1023.461,432.413,-160.150,174.989,50.017,160.490
C04126=1023.474,432.657,-160.201,175.005,50.021,160.494
C04127=1023.487,432.901,-160.252,175.022,50.024,160.497
C04128=1023.500,433.146,-160.303,175.038,50.027,160.501
C04129=1023.513,433.390,-160.354,175.055,50.030,160.505
C04130=1023.525,433.636,-160.406,175.072,50.033,160.509
C04131=1023.538,433.879,-160.457,175.088,50.036,160.512
C04132=1023.551,434.124,-160.508,175.105,50.040,160.516
C04133=1023.564,434.369,-160.560,175.122,50.043,160.520
C04134=1023.577,434.612,-160.611,175.139,50.046,160.524
C04135=1023.591,434.857,-160.662,175.156,50.049,160.528
C04136=1023.603,435.101,-160.714,175.172,50.053,160.531
C04137=1023.617,435.345,-160.766,175.190,50.056,160.535
C04138=1023.630,435.590,-160.817,175.206,50.059,160.539
C04139=1023.644,435.834,-160.869,175.224,50.062,160.543
C04140=1023.660,436.152,-160.936,175.247,50.067,160.548
C04141=1023.678,436.468,-161.003,175.269,50.071,160.553
C04142=1023.695,436.786,-161.071,175.291,50.076,160.558
C04143=1023.713,437.103,-161.138,175.314,50.080,160.563
C04144=1023.726,437.347,-161.190,175.332,50.083,160.567
C04145=1023.740,437.592,-161.242,175.349,50.087,160.571
C04146=1023.753,437.836,-161.294,175.366,50.090,160.575
C04147=1023.766,438.080,-161.347,175.384,50.093,160.579
C04148=1023.780,438.324,-161.399,175.402,50.097,160.584
C04149=1023.794,438.568,-161.452,175.420,50.101,160.587
C04150=1023.807,438.812,-161.504,175.438,50.104,160.592
C04151=1023.820,439.056,-161.557,175.456,50.108,160.596
C04152=1023.834,439.301,-161.609,175.474,50.111,160.600
C04153=1023.848,439.545,-161.662,175.492,50.115,160.604
C04154=1023.862,439.788,-161.714,175.510,50.118,160.608
C04155=1023.875,440.032,-161.768,175.528,50.122,160.612
C04156=1023.889,440.277,-161.820,175.547,50.126,160.617
C04157=1023.903,440.521,-161.872,175.565,50.130,160.621
C04158=1023.918,440.765,-161.925,175.583,50.133,160.625
C04159=1023.931,441.009,-161.978,175.602,50.137,160.629
C04160=1023.946,441.268,-162.034,175.621,50.141,160.634
C04161=1023.961,441.529,-162.091,175.641,50.144,160.638
C04162=1023.976,441.789,-162.148,175.661,50.148,160.643
C04163=1023.991,442.047,-162.205,175.680,50.152,160.647
C04164=1023.596,440.124,-162.120,175.526,50.187,160.632
C04165=1023.583,439.880,-162.067,175.508,50.184,160.628
C04166=1023.569,439.636,-162.014,175.490,50.180,160.624
C04167=1023.555,439.391,-161.962,175.472,50.177,160.620
C04168=1023.541,439.147,-161.909,175.453,50.174,160.615
C04169=1023.528,438.903,-161.856,175.436,50.170,160.611
C04170=1023.514,438.659,-161.804,175.417,50.167,160.607
C04171=1023.501,438.415,-161.752,175.400,50.163,160.603
C04172=1023.487,438.171,-161.700,175.382,50.160,160.599
C04173=1023.474,437.927,-161.647,175.364,50.157,160.595
C04174=1023.460,437.682,-161.594,175.347,50.154,160.591
C04175=1023.446,437.438,-161.542,175.329,50.150,160.587
C04176=1023.433,437.194,-161.491,175.311,50.147,160.583
C04177=1023.419,436.949,-161.439,175.294,50.144,160.579
C04178=1023.406,436.705,-161.387,175.276,50.140,160.575
C04179=1023.393,436.461,-161.335,175.259,50.137,160.571
C04180=1023.379,436.217,-161.283,175.242,50.133,160.567
C04181=1023.366,435.973,-161.231,175.225,50.130,160.564
C04182=1023.353,435.728,-161.180,175.207,50.127,160.560
C04183=1023.340,435.483,-161.128,175.190,50.124,160.556
C04184=1023.327,435.240,-161.076,175.173,50.121,160.552
C04185=1023.314,434.995,-161.025,175.156,50.118,160.548
C04186=1023.300,434.751,-160.973,175.139,50.115,160.544
C04187=1023.287,434.506,-160.922,175.122,50.111,160.540
C04188=1023.274,434.262,-160.871,175.105,50.108,160.537
C04189=1023.261,434.017,-160.819,175.088,50.105,160.533
C04190=1023.248,433.773,-160.769,175.071,50.102,160.529
C04191=1023.235,433.529,-160.717,175.055,50.099,160.525
C04192=1023.222,433.285,-160.666,175.038,50.096,160.522
C04193=1023.209,433.040,-160.615,175.021,50.093,160.518
C04194=1023.197,432.795,-160.563,175.005,50.090,160.514
C04195=1023.184,432.551,-160.512,174.988,50.087,160.511
C04196=1023.170,432.306,-160.462,174.972,50.084,160.507
C04197=1023.158,432.062,-160.411,174.956,50.081,160.503
C04198=1023.144,431.817,-160.360,174.939,50.078,160.500
C04199=1023.132,431.572,-160.310,174.923,50.075,160.496
C04200=1023.119,431.328,-160.259,174.906,50.072,160.492
C04201=1023.106,431.083,-160.208,174.891,50.069,160.489
C04202=1023.093,430.839,-160.158,174.874,50.067,160.485
C04203=1023.081,430.595,-160.107,174.858,50.064,160.482
C04204=1023.068,430.350,-160.057,174.841,50.061,160.478
C04205=1023.054,430.093,-160.005,174.825,50.058,160.475
C04206=1023.042,429.838,-159.952,174.809,50.055,160.471
C04207=1023.028,429.583,-159.899,174.792,50.052,160.467
C04208=1023.015,429.327,-159.847,174.775,50.050,160.464
C04209=1023.003,429.082,-159.797,174.760,50.047,160.460
C04210=1022.991,428.837,-159.747,174.744,50.044,160.457
C04211=1022.978,428.592,-159.697,174.728,50.041,160.453
C04212=1022.966,428.348,-159.647,174.712,50.039,160.450
C04213=1022.954,428.103,-159.596,174.697,50.036,160.447
C04214=1022.941,427.858,-159.546,174.681,50.033,160.443
C04215=1022.928,427.613,-159.497,174.666,50.031,160.440
C04216=1022.916,427.369,-159.447,174.650,50.028,160.436
C04217=1022.900,427.040,-159.380,174.630,50.025,160.432
C04218=1022.884,426.711,-159.313,174.609,50.020,160.427
C04219=1022.867,426.383,-159.247,174.589,50.017,160.423
C04220=1022.852,426.055,-159.180,174.568,50.014,160.419
C04221=1022.839,425.810,-159.131,174.554,50.011,160.416
C04222=1022.827,425.565,-159.081,174.538,50.008,160.412
C04223=1022.816,425.320,-159.032,174.523,50.006,160.409
C04224=1022.803,425.075,-158.982,174.508,50.004,160.406
C04225=1022.791,424.830,-158.934,174.493,50.001,160.402
C04226=1022.779,424.586,-158.884,174.479,49.999,160.399
C04227=1022.767,424.340,-158.835,174.463,49.996,160.396
C04228=1022.755,424.096,-158.787,174.448,49.994,160.393
C04229=1022.743,423.850,-158.737,174.434,49.992,160.390
C04230=1022.731,423.606,-158.689,174.419,49.989,160.387
C04231=1022.719,423.361,-158.640,174.404,49.987,160.383
C04232=1022.707,423.116,-158.590,174.390,49.984,160.380
C04233=1022.695,422.871,-158.542,174.375,49.982,160.377
C04234=1022.684,422.626,-158.493,174.361,49.980,160.374
C04235=1022.672,422.380,-158.444,174.346,49.978,160.371
C04236=1022.660,422.136,-158.396,174.332,49.975,160.368
C04237=1022.649,421.891,-158.347,174.317,49.973,160.365
C04238=1022.637,421.646,-158.299,174.303,49.970,160.362
C04239=1022.625,421.401,-158.250,174.288,49.969,160.359
C04240=1022.614,421.155,-158.202,174.275,49.966,160.356
C04241=1022.602,420.911,-158.153,174.260,49.965,160.353
C04242=1022.590,420.666,-158.105,174.246,49.962,160.350
C04243=1022.579,420.421,-158.057,174.232,49.960,160.347
C04244=1022.567,420.175,-158.009,174.217,49.958,160.344
C04245=1022.555,419.931,-157.960,174.203,49.955,160.341
C04246=1022.544,419.686,-157.913,174.189,49.953,160.338
C04247=1022.532,419.441,-157.865,174.176,49.951,160.335
C04248=1022.521,419.195,-157.817,174.161,49.950,160.332
C04249=1022.509,418.950,-157.769,174.147,49.947,160.329
C04250=1022.498,418.705,-157.721,174.134,49.945,160.326
C04251=1022.486,418.460,-157.673,174.120,49.943,160.324
C04252=1022.474,418.215,-157.625,174.106,49.941,160.321
C04253=1022.463,417.969,-157.578,174.093,49.939,160.318
C04254=1022.451,417.724,-157.530,174.078,49.937,160.315
C04255=1022.441,417.479,-157.482,174.064,49.935,160.312
C04256=1022.429,417.234,-157.434,174.051,49.933,160.309
C04257=1022.418,416.988,-157.387,174.037,49.932,160.307
C04258=1022.406,416.743,-157.339,174.023,49.929,160.304
C04259=1022.395,416.498,-157.293,174.010,49.928,160.301
C04260=1022.384,416.253,-157.244,173.997,49.926,160.298
C04261=1022.373,416.007,-157.197,173.984,49.923,160.295
C04262=1022.362,415.762,-157.149,173.970,49.922,160.293
C04263=1022.351,415.517,-157.102,173.957,49.920,160.290
C04264=1022.340,415.272,-157.055,173.944,49.918,160.287
C04265=1022.329,415.026,-157.007,173.930,49.916,160.285
C04266=1022.318,414.781,-156.961,173.917,49.915,160.282
C04267=1022.306,414.536,-156.914,173.903,49.913,160.279
C04268=1022.295,414.291,-156.867,173.890,49.911,160.277
C04269=1022.284,414.045,-156.820,173.878,49.909,160.274
C04270=1022.273,413.800,-156.774,173.864,49.907,160.271
C04271=1022.262,413.554,-156.726,173.851,49.906,160.268
C04272=1022.251,413.309,-156.679,173.837,49.904,160.266
C04273=1022.240,413.063,-156.632,173.825,49.902,160.263
C04274=1022.229,412.818,-156.586,173.812,49.901,160.261
C04275=1022.218,412.573,-156.540,173.799,49.899,160.258
C04276=1022.207,412.328,-156.493,173.787,49.898,160.256
C04277=1022.192,411.994,-156.429,173.769,49.895,160.252
C04278=1022.178,411.661,-156.367,173.752,49.893,160.248
C04279=1022.163,411.326,-156.303,173.734,49.891,160.245
C04280=1022.149,410.993,-156.240,173.717,49.888,160.241
C04281=1022.138,410.748,-156.194,173.704,49.887,160.239
C04282=1022.127,410.501,-156.147,173.692,49.886,160.237
C04283=1022.116,410.256,-156.101,173.678,49.884,160.234
C04284=1022.105,410.011,-156.055,173.666,49.882,160.231
C04285=1022.094,409.766,-156.008,173.653,49.881,160.229
C04286=1022.084,409.520,-155.962,173.641,49.880,160.227
C04287=1022.074,409.274,-155.916,173.628,49.878,160.224
C04288=1022.063,409.029,-155.870,173.616,49.877,160.222
C04289=1022.053,408.783,-155.824,173.604,49.875,160.219
C04290=1022.041,408.538,-155.779,173.591,49.874,160.217
C04291=1022.031,408.292,-155.733,173.579,49.873,160.214
C04292=1022.020,408.047,-155.687,173.567,49.871,160.212
C04293=1022.010,407.802,-155.641,173.554,49.870,160.210
C04294=1021.999,407.556,-155.595,173.542,49.868,160.207
C04295=1021.989,407.310,-155.550,173.531,49.867,160.205
C04296=1021.978,407.065,-155.505,173.518,49.866,160.202
C04297=1021.967,406.819,-155.459,173.506,49.864,160.200
C04298=1021.957,406.574,-155.414,173.494,49.863,160.198
C04299=1021.947,406.328,-155.368,173.482,49.862,160.195
C04300=1021.936,406.082,-155.322,173.469,49.861,160.193
C04301=1021.926,405.836,-155.277,173.457,49.860,160.191
C04302=1021.915,405.592,-155.232,173.445,49.858,160.188
C04303=1021.905,405.345,-155.187,173.434,49.857,160.186
C04304=1021.894,405.100,-155.141,173.422,49.856,160.184
C04305=1021.884,404.854,-155.096,173.410,49.854,160.182
C04306=1021.874,404.608,-155.051,173.398,49.853,160.179
C04307=1021.863,404.363,-155.006,173.386,49.853,160.177
C04308=1021.853,404.117,-154.961,173.374,49.851,160.175
C04309=1021.843,403.872,-154.916,173.362,49.850,160.173
C04310=1021.833,403.625,-154.871,173.350,49.849,160.170
C04311=1021.823,403.381,-154.825,173.339,49.848,160.168
C04312=1021.813,403.134,-154.780,173.327,49.847,160.166
C04313=1021.802,402.889,-154.736,173.315,49.846,160.164
C04314=1021.792,402.644,-154.691,173.303,49.845,160.161
C04315=1021.782,402.397,-154.646,173.292,49.844,160.159
C04316=1021.772,402.152,-154.601,173.281,49.842,160.157
C04317=1021.763,401.906,-154.556,173.270,49.842,160.155
C04318=1021.752,401.660,-154.511,173.258,49.841,160.153
C04319=1021.742,401.415,-154.467,173.247,49.840,160.151
C04320=1021.732,401.170,-154.422,173.235,49.839,160.148
C04321=1021.723,400.923,-154.378,173.223,49.838,160.146
C04322=1021.712,400.677,-154.333,173.212,49.837,160.144
C04323=1021.702,400.432,-154.289,173.200,49.836,160.142
C04324=1021.693,400.186,-154.245,173.190,49.835,160.140
C04325=1021.683,399.940,-154.200,173.178,49.834,160.138
C04326=1021.672,399.695,-154.155,173.167,49.833,160.136
C04327=1021.663,399.449,-154.111,173.155,49.832,160.134
C04328=1021.653,399.203,-154.067,173.144,49.832,160.132
C04329=1021.643,398.957,-154.023,173.133,49.830,160.130
C04330=1021.633,398.711,-153.979,173.122,49.830,160.128
C04331=1021.623,398.466,-153.934,173.111,49.829,160.125
C04332=1021.613,398.219,-153.890,173.099,49.828,160.123
C04333=1021.604,397.973,-153.846,173.089,49.827,160.121
C04334=1021.594,397.727,-153.803,173.077,49.827,160.119
C04335=1021.584,397.482,-153.758,173.066,49.826,160.117
C04336=1021.574,397.236,-153.714,173.056,49.825,160.115
C04337=1021.562,396.925,-153.659,173.042,49.824,160.113
C04338=1021.549,396.614,-153.604,173.028,49.823,160.110
C04339=1021.537,396.303,-153.548,173.014,49.822,160.108
C04340=1021.525,395.992,-153.493,173.000,49.822,160.105
C04341=1021.514,395.746,-153.449,172.990,49.821,160.104
C04342=1021.506,395.500,-153.406,172.979,49.821,160.102
C04343=1021.496,395.255,-153.363,172.967,49.820,160.100
C04344=1021.486,395.009,-153.319,172.957,49.819,160.098
C04345=1021.476,394.763,-153.275,172.946,49.819,160.096
C04346=1021.466,394.516,-153.232,172.936,49.818,160.094
C04347=1021.458,394.271,-153.189,172.924,49.818,160.092
C04348=1021.447,394.025,-153.145,172.914,49.817,160.090
C04349=1021.438,393.778,-153.102,172.903,49.817,160.088
C04350=1021.429,393.533,-153.059,172.893,49.816,160.086
C04351=1021.419,393.287,-153.016,172.882,49.816,160.084
C04352=1021.410,393.040,-152.972,172.871,49.815,160.082
C04353=1021.400,392.795,-152.929,172.862,49.814,160.081
C04354=1021.391,392.549,-152.885,172.850,49.814,160.079
C04355=1021.382,392.303,-152.843,172.840,49.814,160.077
C04356=1021.372,392.056,-152.800,172.829,49.813,160.075
C04357=1021.362,391.811,-152.756,172.819,49.813,160.073
C04358=1021.353,391.565,-152.713,172.809,49.812,160.072
C04359=1021.343,391.318,-152.671,172.798,49.812,160.070
C04360=1021.334,391.072,-152.628,172.788,49.811,160.068
C04361=1021.324,390.826,-152.585,172.778,49.811,160.066
C04362=1021.315,390.580,-152.543,172.767,49.811,160.064
C04363=1021.306,390.333,-152.500,172.757,49.810,160.063
C04364=1021.296,390.088,-152.456,172.747,49.810,160.061
C04365=1021.287,389.842,-152.415,172.736,49.810,160.059
C04366=1021.278,389.595,-152.372,172.726,49.810,160.057
C04367=1021.269,389.349,-152.329,172.716,49.810,160.056
C04368=1021.260,389.104,-152.286,172.706,49.809,160.054
C04369=1021.250,388.857,-152.244,172.695,49.809,160.052
C04370=1021.241,388.611,-152.201,172.685,49.809,160.050
C04371=1021.231,388.366,-152.159,172.675,49.808,160.049
C04372=1021.223,388.118,-152.116,172.666,49.808,160.047
C04373=1021.213,387.873,-152.074,172.656,49.808,160.045
C04374=1021.204,387.627,-152.031,172.645,49.808,160.044
C04375=1021.195,387.380,-151.989,172.635,49.808,160.042
C04376=1021.185,387.134,-151.947,172.625,49.807,160.040
C04377=1021.177,386.888,-151.905,172.616,49.808,160.039
C04378=1021.167,386.642,-151.863,172.606,49.807,160.037
C04379=1021.158,386.396,-151.821,172.596,49.807,160.035
C04380=1021.149,386.150,-151.778,172.585,49.807,160.034
C04381=1021.140,385.903,-151.736,172.575,49.807,160.032
C04382=1021.130,385.657,-151.694,172.566,49.807,160.030
C04383=1021.121,385.411,-151.652,172.556,49.807,160.029
C04384=1021.112,385.164,-151.610,172.546,49.807,160.027
C04385=1021.104,384.918,-151.569,172.536,49.807,160.026
C04386=1021.095,384.672,-151.527,172.526,49.807,160.024
C04387=1021.086,384.425,-151.485,172.517,49.807,160.022
C04388=1021.077,384.179,-151.444,172.507,49.807,160.021
C04389=1021.067,383.933,-151.402,172.497,49.807,160.019
C04390=1021.058,383.687,-151.360,172.488,49.807,160.018
C04391=1021.049,383.441,-151.318,172.478,49.807,160.016
C04392=1021.040,383.194,-151.277,172.469,49.807,160.015
C04393=1021.031,382.947,-151.236,172.459,49.807,160.013
C04394=1021.022,382.701,-151.194,172.449,49.807,160.011
C04395=1021.013,382.455,-151.153,172.440,49.808,160.010
C04396=1021.004,382.209,-151.111,172.430,49.808,160.009
C04397=1020.994,381.934,-151.065,172.419,49.808,160.007
C04398=1020.984,381.661,-151.019,172.408,49.808,160.005
C04399=1020.975,381.387,-150.973,172.398,49.809,160.003
C04400=1020.964,381.113,-150.927,172.387,49.809,160.002
C04401=1020.956,380.867,-150.886,172.379,49.809,160.000
C04402=1020.947,380.621,-150.844,172.369,49.809,159.999
C04403=1020.938,380.374,-150.804,172.360,49.809,159.997
C04404=1020.929,380.128,-150.762,172.350,49.810,159.996
C04405=1020.920,379.882,-150.721,172.341,49.810,159.994
C04406=1020.912,379.635,-150.680,172.331,49.810,159.993
C04407=1020.903,379.389,-150.638,172.321,49.811,159.991
C04408=1020.894,379.142,-150.597,172.313,49.811,159.990
C04409=1020.885,378.896,-150.557,172.303,49.811,159.989
C04410=1020.876,378.649,-150.515,172.294,49.811,159.987
C04411=1020.868,378.403,-150.475,172.284,49.812,159.986
C04412=1020.859,378.157,-150.433,172.275,49.812,159.984
C04413=1020.851,377.910,-150.392,172.266,49.812,159.983
C04414=1020.842,377.664,-150.352,172.257,49.813,159.981
C04415=1020.833,377.417,-150.311,172.248,49.813,159.980
C04416=1020.825,377.171,-150.270,172.238,49.813,159.979
C04417=1020.816,376.924,-150.229,172.230,49.813,159.977
C04418=1020.808,376.678,-150.188,172.221,49.814,159.976
C04419=1020.800,376.431,-150.147,172.211,49.814,159.974
C04420=1020.791,376.185,-150.107,172.202,49.815,159.973
C04421=1020.782,375.938,-150.066,172.193,49.815,159.972
C04422=1020.774,375.692,-150.026,172.184,49.816,159.970
C04423=1020.765,375.445,-149.985,172.175,49.816,159.969
C04424=1020.756,375.199,-149.945,172.167,49.817,159.968
C04425=1020.748,374.952,-149.904,172.157,49.817,159.966
C04426=1020.739,374.705,-149.865,172.148,49.818,159.965
C04427=1020.731,374.458,-149.824,172.139,49.818,159.964
C04428=1020.722,374.212,-149.783,172.130,49.819,159.962
C04429=1020.714,373.966,-149.743,172.121,49.820,159.961
C04430=1020.705,373.719,-149.703,172.112,49.820,159.960
C04431=1020.697,373.473,-149.663,172.104,49.821,159.958
C04432=1020.688,373.225,-149.623,172.095,49.822,159.957
C04433=1020.680,372.979,-149.582,172.086,49.822,159.956
C04434=1020.671,372.733,-149.542,172.077,49.823,159.955
C04435=1020.663,372.486,-149.502,172.068,49.823,159.953
C04436=1020.654,372.239,-149.462,172.060,49.824,159.952
C04437=1020.646,371.993,-149.422,172.050,49.825,159.951
C04438=1020.637,371.747,-149.382,172.042,49.825,159.950
C04439=1020.629,371.500,-149.343,172.033,49.826,159.948
C04440=1020.620,371.252,-149.302,172.024,49.827,159.947
C04441=1020.612,371.006,-149.262,172.016,49.828,159.946
C04442=1020.604,370.759,-149.222,172.007,49.829,159.945
C04443=1020.596,370.513,-149.183,171.999,49.829,159.943
C04444=1020.588,370.267,-149.142,171.990,49.830,159.942
C04445=1020.579,370.020,-149.103,171.981,49.830,159.941
C04446=1020.571,369.773,-149.063,171.972,49.831,159.940
C04447=1020.562,369.526,-149.023,171.964,49.832,159.938
C04448=1020.554,369.280,-148.983,171.955,49.833,159.937
C04449=1020.546,369.033,-148.943,171.947,49.833,159.936
C04450=1020.538,368.786,-148.904,171.938,49.835,159.935
C04451=1020.530,368.539,-148.864,171.930,49.835,159.934
C04452=1020.522,368.293,-148.824,171.921,49.836,159.933
C04453=1020.513,368.046,-148.785,171.913,49.837,159.931
C04454=1020.505,367.799,-148.746,171.905,49.838,159.930
C04455=1020.497,367.552,-148.706,171.896,49.839,159.929
C04456=1020.489,367.306,-148.666,171.888,49.839,159.928
C04457=1020.480,367.054,-148.627,171.879,49.841,159.927
C04458=1020.473,366.803,-148.587,171.870,49.842,159.926
C04459=1020.464,366.551,-148.547,171.862,49.843,159.925
C04460=1020.455,366.299,-148.507,171.853,49.844,159.923
C04461=1020.447,366.053,-148.467,171.845,49.845,159.922
C04462=1020.439,365.806,-148.429,171.836,49.846,159.921
C04463=1020.430,365.559,-148.389,171.828,49.847,159.920
C04464=1020.422,365.313,-148.350,171.820,49.847,159.919
C04465=1020.414,365.066,-148.312,171.811,49.849,159.918
C04466=1020.406,364.819,-148.273,171.804,49.850,159.917
C04467=1020.398,364.572,-148.233,171.794,49.851,159.916
C04468=1020.390,364.325,-148.194,171.787,49.852,159.915
C04469=1020.382,364.078,-148.155,171.779,49.853,159.914
C04470=1020.374,363.832,-148.116,171.770,49.854,159.912
C04471=1020.366,363.585,-148.078,171.762,49.855,159.911
C04472=1020.357,363.338,-148.039,171.754,49.856,159.910
C04473=1020.349,363.091,-148.000,171.745,49.858,159.909
C04474=1020.342,362.844,-147.961,171.738,49.859,159.908
C04475=1020.334,362.598,-147.922,171.730,49.860,159.907
C04476=1020.326,362.350,-147.883,171.722,49.861,159.906
C04477=1020.318,362.104,-147.845,171.713,49.862,159.905
C04478=1020.310,361.857,-147.806,171.705,49.863,159.904
C04479=1020.302,361.610,-147.767,171.697,49.864,159.903
C04480=1020.294,361.364,-147.729,171.689,49.866,159.902
C04481=1020.286,361.116,-147.690,171.681,49.867,159.901
C04482=1020.278,360.869,-147.651,171.673,49.868,159.900
C04483=1020.271,360.622,-147.613,171.665,49.869,159.899
C04484=1020.263,360.375,-147.574,171.657,49.871,159.898
C04485=1020.255,360.129,-147.536,171.649,49.872,159.897
C04486=1020.247,359.882,-147.497,171.641,49.873,159.896
C04487=1020.239,359.635,-147.458,171.633,49.874,159.895
C04488=1020.231,359.388,-147.420,171.625,49.876,159.894
C04489=1020.224,359.141,-147.382,171.617,49.877,159.893
C04490=1020.216,358.894,-147.344,171.609,49.879,159.892
C04491=1020.208,358.647,-147.305,171.602,49.880,159.891
C04492=1020.200,358.400,-147.267,171.594,49.881,159.890
C04493=1020.192,358.154,-147.229,171.585,49.882,159.889
C04494=1020.184,357.906,-147.191,171.578,49.884,159.888
C04495=1020.176,357.660,-147.153,171.570,49.885,159.887
C04496=1020.168,357.412,-147.114,171.562,49.886,159.886
C04497=1020.161,357.165,-147.077,171.555,49.888,159.886
C04498=1020.153,356.918,-147.038,171.546,49.890,159.885
C04499=1020.144,356.672,-147.000,171.539,49.891,159.884
C04500=1020.137,356.425,-146.963,171.531,49.893,159.883
C04501=1020.129,356.177,-146.924,171.524,49.894,159.882
C04502=1020.122,355.930,-146.887,171.516,49.895,159.881
C04503=1020.114,355.684,-146.849,171.508,49.897,159.880
C04504=1020.106,355.436,-146.811,171.500,49.899,159.879
C04505=1020.098,355.190,-146.773,171.492,49.900,159.878
C04506=1020.091,354.943,-146.736,171.484,49.902,159.877
C04507=1020.083,354.695,-146.698,171.477,49.903,159.877
C04508=1020.075,354.448,-146.659,171.469,49.904,159.876
C04509=1020.067,354.201,-146.622,171.462,49.906,159.875
C04510=1020.060,353.955,-146.584,171.454,49.908,159.874
C04511=1020.052,353.707,-146.546,171.447,49.909,159.873
C04512=1020.044,353.460,-146.509,171.438,49.911,159.872
C04513=1020.037,353.214,-146.472,171.431,49.913,159.871
C04514=1020.029,352.969,-146.434,171.424,49.915,159.871
C04515=1020.022,352.724,-146.397,171.416,49.916,159.870
C04516=1020.014,352.477,-146.360,171.408,49.918,159.869
C04517=1020.007,352.232,-146.323,171.401,49.919,159.868
C04518=1019.999,351.986,-146.286,171.394,49.921,159.867
C04519=1019.991,351.741,-146.249,171.386,49.923,159.866
C04520=1019.984,351.495,-146.211,171.379,49.925,159.866
C04521=1019.976,351.248,-146.173,171.371,49.926,159.865
C04522=1019.968,351.001,-146.136,171.364,49.928,159.864
C04523=1019.961,350.753,-146.100,171.357,49.930,159.863
C04524=1019.953,350.506,-146.063,171.349,49.932,159.863
C04525=1019.946,350.259,-146.025,171.342,49.933,159.862
C04526=1019.938,350.012,-145.988,171.334,49.935,159.861
C04527=1019.930,349.765,-145.951,171.327,49.937,159.860
C04528=1019.923,349.518,-145.913,171.320,49.939,159.859
C04529=1019.915,349.271,-145.876,171.312,49.940,159.859
C04530=1019.908,349.024,-145.839,171.305,49.942,159.858
C04531=1019.901,348.776,-145.802,171.297,49.944,159.857
C04532=1019.893,348.529,-145.765,171.290,49.946,159.856
C04533=1019.886,348.282,-145.727,171.283,49.947,159.856
C04534=1019.878,348.035,-145.691,171.275,49.949,159.855
C04535=1019.871,347.788,-145.654,171.268,49.952,159.854
C04536=1019.863,347.541,-145.617,171.261,49.953,159.853
C04537=1019.856,347.293,-145.580,171.253,49.955,159.853
C04538=1019.848,347.046,-145.543,171.246,49.957,159.852
C04539=1019.842,346.799,-145.507,171.239,49.959,159.851
C04540=1019.834,346.552,-145.470,171.232,49.961,159.850
C04541=1019.826,346.305,-145.433,171.224,49.963,159.850
C04542=1019.819,346.058,-145.396,171.217,49.965,159.849
C04543=1019.811,345.810,-145.360,171.210,49.967,159.848
C04544=1019.803,345.563,-145.323,171.203,49.969,159.848
C04545=1019.796,345.316,-145.286,171.195,49.971,159.847
C04546=1019.789,345.069,-145.250,171.188,49.973,159.846
C04547=1019.781,344.822,-145.214,171.181,49.975,159.846
C04548=1019.774,344.575,-145.176,171.174,49.977,159.845
C04549=1019.766,344.327,-145.140,171.167,49.979,159.844
C04550=1019.759,344.080,-145.104,171.160,49.982,159.844
C04551=1019.752,343.833,-145.067,171.152,49.983,159.843
C04552=1019.744,343.586,-145.031,171.145,49.986,159.842
C04553=1019.737,343.338,-144.994,171.138,49.987,159.841
C04554=1019.730,343.091,-144.958,171.131,49.990,159.841
C04555=1019.723,342.844,-144.922,171.123,49.992,159.840
C04556=1019.715,342.596,-144.885,171.117,49.994,159.840
C04557=1019.707,342.349,-144.849,171.110,49.996,159.839
C04558=1019.701,342.102,-144.813,171.103,49.998,159.838
C04559=1019.693,341.854,-144.777,171.096,50.000,159.838
C04560=1019.686,341.607,-144.740,171.089,50.003,159.837
C04561=1019.679,341.360,-144.704,171.082,50.005,159.836
C04562=1019.672,341.112,-144.668,171.074,50.007,159.836
C04563=1019.665,340.866,-144.632,171.067,50.009,159.835
C04564=1019.657,340.618,-144.596,171.060,50.011,159.834
C04565=1019.649,340.371,-144.559,171.054,50.013,159.834
C04566=1019.643,340.124,-144.523,171.047,50.016,159.833
C04567=1019.635,339.876,-144.487,171.040,50.018,159.833
C04568=1019.628,339.629,-144.452,171.033,50.021,159.832
C04569=1019.621,339.382,-144.415,171.026,50.022,159.831
C04570=1019.614,339.135,-144.380,171.019,50.025,159.831
C04571=1019.606,338.887,-144.343,171.012,50.027,159.830
C04572=1019.599,338.640,-144.308,171.005,50.030,159.830
C04573=1019.592,338.393,-144.272,170.999,50.032,159.829
C04574=1019.585,338.146,-144.236,170.992,50.034,159.829
C04575=1019.578,337.898,-144.201,170.985,50.037,159.828
C04576=1019.570,337.651,-144.165,170.978,50.039,159.828
C04577=1019.563,337.404,-144.129,170.971,50.042,159.827
C04578=1019.556,337.157,-144.094,170.964,50.044,159.826
C04579=1019.549,336.909,-144.058,170.958,50.046,159.826
C04580=1019.542,336.662,-144.022,170.951,50.049,159.825
C04581=1019.535,336.415,-143.987,170.944,50.051,159.825
C04582=1019.527,336.167,-143.951,170.937,50.054,159.824
C04583=1019.520,335.921,-143.915,170.930,50.056,159.824
C04584=1019.513,335.672,-143.880,170.923,50.059,159.823
C04585=1019.506,335.425,-143.845,170.917,50.061,159.823
C04586=1019.499,335.178,-143.809,170.910,50.063,159.822
C04587=1019.492,334.930,-143.773,170.904,50.066,159.822
C04588=1019.485,334.683,-143.738,170.897,50.069,159.821
C04589=1019.478,334.436,-143.702,170.890,50.071,159.820
C04590=1019.471,334.189,-143.667,170.884,50.074,159.820
C04591=1019.464,333.941,-143.632,170.877,50.076,159.820
C04592=1019.457,333.693,-143.596,170.870,50.078,159.819
C04593=1019.450,333.447,-143.561,170.863,50.081,159.819
C04594=1019.443,333.199,-143.525,170.856,50.084,159.818
C04595=1019.436,332.951,-143.490,170.851,50.086,159.818
C04596=1019.428,332.704,-143.455,170.844,50.089,159.817
C04597=1019.421,332.457,-143.420,170.837,50.092,159.817
C04598=1019.415,332.209,-143.385,170.830,50.094,159.816
C04599=1019.407,331.961,-143.350,170.823,50.097,159.816
C04600=1019.400,331.714,-143.315,170.817,50.099,159.815
C04601=1019.393,331.467,-143.280,170.811,50.102,159.815
C04602=1019.386,331.220,-143.245,170.804,50.105,159.814
C04603=1019.379,330.973,-143.210,170.797,50.108,159.814
C04604=1019.371,330.724,-143.175,170.790,50.111,159.814
C04605=1019.365,330.477,-143.140,170.784,50.113,159.813
C04606=1019.358,330.230,-143.105,170.778,50.116,159.813
C04607=1019.351,329.982,-143.071,170.771,50.119,159.812
C04608=1019.344,329.735,-143.036,170.764,50.121,159.812
C04609=1019.337,329.487,-143.000,170.758,50.124,159.811
C04610=1019.330,329.240,-142.965,170.752,50.127,159.811
C04611=1019.323,328.993,-142.931,170.745,50.130,159.811
C04612=1019.316,328.745,-142.896,170.738,50.132,159.810
C04613=1019.310,328.498,-142.861,170.732,50.135,159.810
C04614=1019.302,328.250,-142.827,170.726,50.138,159.809
C04615=1019.295,328.002,-142.792,170.719,50.141,159.809
C04616=1019.288,327.754,-142.757,170.712,50.143,159.808
C04617=1019.282,327.507,-142.722,170.706,50.146,159.808
C04618=1019.275,327.260,-142.688,170.700,50.149,159.808
C04619=1019.268,327.013,-142.653,170.693,50.152,159.807
C04620=1019.261,326.765,-142.618,170.688,50.155,159.807
C04621=1019.254,326.518,-142.584,170.681,50.158,159.806
C04622=1019.247,326.270,-142.549,170.674,50.161,159.806
C04623=1019.240,326.023,-142.515,170.668,50.164,159.806
C04624=1019.233,325.775,-142.481,170.662,50.167,159.805
C04625=1019.226,325.528,-142.447,170.655,50.170,159.805
C04626=1019.219,325.280,-142.412,170.649,50.173,159.805
C04627=1019.212,325.032,-142.379,170.642,50.176,159.804
C04628=1019.205,324.785,-142.345,170.636,50.179,159.804
C04629=1019.198,324.537,-142.310,170.630,50.182,159.804
C04630=1019.191,324.290,-142.276,170.623,50.185,159.803
C04631=1019.183,324.042,-142.242,170.617,50.188,159.803
C04632=1019.176,323.794,-142.208,170.610,50.191,159.803
C04633=1019.170,323.546,-142.174,170.605,50.195,159.802
C04634=1019.163,323.300,-142.139,170.598,50.198,159.802
C04635=1019.156,323.052,-142.106,170.592,50.201,159.802
C04636=1019.149,322.805,-142.072,170.585,50.204,159.801
C04637=1019.142,322.553,-142.037,170.580,50.207,159.801
C04638=1019.135,322.302,-142.003,170.573,50.210,159.801
C04639=1019.128,322.050,-141.969,170.566,50.213,159.800
C04640=1019.121,321.799,-141.934,170.560,50.217,159.800
C04641=1019.114,321.551,-141.900,170.554,50.220,159.800
C04642=1019.108,321.304,-141.866,170.548,50.222,159.799
C04643=1019.101,321.056,-141.832,170.542,50.226,159.799
C04644=1019.093,320.808,-141.799,170.535,50.229,159.799
C04645=1019.086,320.561,-141.765,170.529,50.233,159.799
C04646=1019.080,320.314,-141.731,170.523,50.236,159.798
C04647=1019.073,320.066,-141.697,170.517,50.239,159.798
C04648=1019.066,319.818,-141.663,170.510,50.242,159.798
C04649=1019.059,319.571,-141.630,170.505,50.245,159.797
C04650=1019.053,319.323,-141.595,170.498,50.249,159.797
C04651=1019.046,319.076,-141.561,170.492,50.252,159.797
C04652=1019.039,318.828,-141.529,170.486,50.255,159.797
C04653=1019.032,318.580,-141.495,170.480,50.259,159.797
C04654=1019.026,318.332,-141.460,170.473,50.262,159.796
C04655=1019.019,318.085,-141.427,170.468,50.265,159.796
C04656=1019.012,317.838,-141.393,170.462,50.268,159.796
C04657=1019.006,317.590,-141.360,170.455,50.272,159.796
C04658=1018.999,317.342,-141.326,170.450,50.274,159.795
C04659=1018.992,317.095,-141.292,170.443,50.278,159.795
C04660=1018.986,316.847,-141.259,170.437,50.282,159.795
C04661=1018.978,316.599,-141.225,170.431,50.285,159.795
C04662=1018.972,316.352,-141.192,170.425,50.288,159.794
C04663=1018.966,316.104,-141.158,170.419,50.292,159.794
C04664=1018.959,315.857,-141.125,170.413,50.295,159.794
C04665=1018.952,315.609,-141.091,170.407,50.298,159.794
C04666=1018.946,315.361,-141.058,170.401,50.302,159.793
C04667=1018.940,315.114,-141.024,170.396,50.305,159.793
C04668=1018.933,314.866,-140.991,170.389,50.308,159.793
C04669=1018.926,314.619,-140.958,170.383,50.312,159.793
C04670=1018.919,314.370,-140.925,170.377,50.315,159.793
C04671=1018.913,314.123,-140.891,170.371,50.319,159.792
C04672=1018.907,313.875,-140.857,170.366,50.322,159.792
C04673=1018.900,313.628,-140.824,170.359,50.325,159.792
C04674=1018.894,313.380,-140.791,170.353,50.329,159.792
C04675=1018.886,313.133,-140.757,170.348,50.332,159.792
C04676=1018.881,312.885,-140.724,170.341,50.336,159.791
C04677=1018.875,312.637,-140.691,170.335,50.340,159.791
C04678=1018.867,312.389,-140.657,170.330,50.343,159.791
C04679=1018.861,312.142,-140.625,170.324,50.347,159.791
C04680=1018.855,311.895,-140.591,170.318,50.350,159.791
C04681=1018.848,311.646,-140.558,170.312,50.354,159.791
C04682=1018.842,311.399,-140.525,170.305,50.357,159.790
C04683=1018.835,311.152,-140.491,170.300,50.360,159.790
C04684=1018.829,310.904,-140.459,170.294,50.364,159.790
C04685=1018.823,310.656,-140.425,170.289,50.367,159.790
C04686=1018.817,310.408,-140.392,170.282,50.371,159.790
C04687=1018.810,310.161,-140.359,170.277,50.374,159.789
C04688=1018.804,309.913,-140.326,170.271,50.378,159.789
C04689=1018.797,309.665,-140.293,170.265,50.382,159.789
C04690=1018.791,309.417,-140.260,170.260,50.386,159.789
C04691=1018.784,309.170,-140.228,170.253,50.390,159.789
C04692=1018.777,308.923,-140.195,170.248,50.394,159.789
C04693=1018.770,308.675,-140.163,170.242,50.397,159.789
C04694=1018.764,308.429,-140.131,170.236,50.401,159.789
C04695=1018.757,308.182,-140.098,170.230,50.405,159.789
C04696=1018.750,307.935,-140.066,170.225,50.409,159.788
C04697=1018.744,307.688,-140.034,170.219,50.412,159.788
C04698=1018.737,307.441,-140.002,170.213,50.417,159.788
C04699=1018.730,307.195,-139.969,170.208,50.420,159.788
C04700=1018.724,306.948,-139.937,170.201,50.424,159.788
C04701=1018.717,306.700,-139.904,170.195,50.428,159.788
C04702=1018.711,306.452,-139.872,170.190,50.431,159.788
C04703=1018.704,306.204,-139.840,170.184,50.436,159.788
C04704=1018.697,305.957,-139.807,170.178,50.440,159.788
C04705=1018.691,305.709,-139.775,170.173,50.444,159.788
C04706=1018.684,305.461,-139.743,170.167,50.447,159.788
C04707=1018.677,305.213,-139.710,170.161,50.452,159.788
C04708=1018.671,304.965,-139.679,170.156,50.455,159.787
C04709=1018.664,304.718,-139.646,170.150,50.459,159.787
C04710=1018.657,304.470,-139.614,170.144,50.463,159.787
C04711=1018.651,304.222,-139.582,170.139,50.467,159.787
C04712=1018.645,303.974,-139.549,170.133,50.471,159.787
C04713=1018.638,303.727,-139.518,170.127,50.475,159.787
C04714=1018.632,303.479,-139.485,170.122,50.479,159.787
C04715=1018.625,303.231,-139.453,170.116,50.483,159.787
C04716=1018.619,302.983,-139.421,170.110,50.487,159.787
C04717=1018.612,302.736,-139.389,170.105,50.491,159.787
C04718=1018.606,302.488,-139.357,170.099,50.495,159.787
C04719=1018.600,302.240,-139.325,170.093,50.499,159.787
C04720=1018.593,301.992,-139.292,170.088,50.503,159.787
C04721=1018.587,301.744,-139.260,170.082,50.508,159.787
C04722=1018.580,301.496,-139.229,170.077,50.511,159.787
C04723=1018.574,301.249,-139.196,170.071,50.515,159.787
C04724=1018.567,301.001,-139.165,170.065,50.520,159.787
C04725=1018.561,300.753,-139.133,170.060,50.524,159.787
C04726=1018.555,300.505,-139.100,170.054,50.527,159.787
C04727=1018.548,300.257,-139.069,170.048,50.532,159.787
C04728=1018.542,300.009,-139.037,170.043,50.536,159.787
C04729=1018.535,299.762,-139.004,170.037,50.540,159.787
C04730=1018.529,299.513,-138.972,170.032,50.544,159.787
C04731=1018.523,299.266,-138.941,170.026,50.548,159.787
C04732=1018.517,299.018,-138.909,170.020,50.552,159.787
C04733=1018.511,298.770,-138.877,170.015,50.556,159.787
C04734=1018.504,298.523,-138.845,170.009,50.561,159.787
C04735=1018.498,298.274,-138.813,170.004,50.565,159.787
C04736=1018.491,298.026,-138.782,169.999,50.569,159.787
C04737=1018.485,297.778,-138.750,169.993,50.574,159.787
C04738=1018.479,297.531,-138.719,169.988,50.578,159.787
C04739=1018.473,297.283,-138.686,169.982,50.582,159.787
C04740=1018.466,297.035,-138.654,169.976,50.586,159.787
C04741=1018.460,296.787,-138.622,169.971,50.590,159.787
C04742=1018.454,296.539,-138.590,169.966,50.595,159.787
C04743=1018.448,296.292,-138.559,169.961,50.599,159.787
C04744=1018.442,296.044,-138.527,169.955,50.603,159.787
C04745=1018.436,295.796,-138.496,169.950,50.607,159.787
C04746=1018.430,295.548,-138.464,169.944,50.612,159.787
C04747=1018.423,295.300,-138.433,169.938,50.616,159.787
C04748=1018.417,295.052,-138.401,169.933,50.620,159.787
C04749=1018.411,294.804,-138.369,169.927,50.624,159.787
C04750=1018.405,294.557,-138.338,169.923,50.628,159.787
C04751=1018.399,294.308,-138.306,169.917,50.633,159.787
C04752=1018.393,294.061,-138.274,169.911,50.637,159.787
C04753=1018.387,293.822,-138.244,169.906,50.641,159.787
C04754=1018.381,293.584,-138.214,169.901,50.645,159.787
C04755=1018.376,293.346,-138.183,169.895,50.650,159.787
C04756=1018.370,293.108,-138.153,169.890,50.654,159.788
C04757=1018.363,292.870,-138.123,169.886,50.658,159.788
C04758=1018.358,292.632,-138.093,169.880,50.663,159.788
C04759=1018.351,292.394,-138.063,169.875,50.667,159.788
C04760=1018.346,292.156,-138.033,169.870,50.671,159.788
C04761=1018.340,291.909,-138.002,169.864,50.675,159.788
C04762=1018.333,291.661,-137.971,169.859,50.680,159.788
C04763=1018.326,291.413,-137.940,169.854,50.684,159.788
C04764=1018.320,291.165,-137.909,169.849,50.689,159.788
C04765=1018.314,290.917,-137.878,169.843,50.694,159.788
C04766=1018.308,290.669,-137.846,169.838,50.698,159.788
C04767=1018.302,290.421,-137.816,169.832,50.703,159.789
C04768=1018.295,290.173,-137.784,169.827,50.707,159.789
C04769=1018.289,289.925,-137.754,169.822,50.712,159.789
C04770=1018.283,289.677,-137.722,169.816,50.716,159.789
C04771=1018.277,289.429,-137.692,169.812,50.721,159.789
C04772=1018.271,289.181,-137.661,169.806,50.725,159.789
C04773=1018.264,288.933,-137.630,169.800,50.730,159.789
C04774=1018.258,288.685,-137.600,169.796,50.735,159.790
C04775=1018.251,288.437,-137.568,169.790,50.740,159.790
C04776=1018.245,288.189,-137.538,169.785,50.745,159.790
C04777=1018.239,287.941,-137.507,169.780,50.749,159.790
C04778=1018.233,287.694,-137.476,169.774,50.754,159.790
C04779=1018.226,287.445,-137.445,169.769,50.759,159.790
C04780=1018.221,287.197,-137.415,169.764,50.763,159.790
C04781=1018.214,286.949,-137.383,169.759,50.768,159.791
C04782=1018.208,286.702,-137.353,169.753,50.773,159.791
C04783=1018.202,286.453,-137.322,169.748,50.777,159.791
C04784=1018.196,286.205,-137.292,169.743,50.782,159.791
C04785=1018.189,285.957,-137.261,169.737,50.787,159.791
C04786=1018.183,285.710,-137.230,169.733,50.792,159.792
C04787=1018.177,285.461,-137.200,169.727,50.796,159.792
C04788=1018.171,285.213,-137.169,169.722,50.801,159.792
C04789=1018.165,284.965,-137.139,169.717,50.806,159.792
C04790=1018.159,284.717,-137.108,169.712,50.811,159.792
C04791=1018.153,284.469,-137.078,169.706,50.816,159.792
C04792=1018.147,284.221,-137.047,169.701,50.820,159.792
C04793=1018.141,283.973,-137.017,169.696,50.825,159.793
C04794=1018.134,283.725,-136.987,169.690,50.830,159.793
C04795=1018.128,283.477,-136.956,169.686,50.835,159.793
C04796=1018.122,283.229,-136.926,169.680,50.840,159.793
C04797=1018.116,282.980,-136.895,169.675,50.845,159.794
C04798=1018.109,282.733,-136.865,169.670,50.850,159.794
C04799=1018.103,282.485,-136.835,169.665,50.855,159.794
C04800=1018.097,282.236,-136.804,169.660,50.860,159.794
C04801=1018.091,281.989,-136.774,169.654,50.865,159.794
C04802=1018.084,281.741,-136.744,169.650,50.870,159.795
C04803=1018.078,281.492,-136.714,169.644,50.875,159.795
C04804=1018.073,281.244,-136.684,169.639,50.880,159.795
C04805=1018.067,280.996,-136.654,169.634,50.885,159.795
C04806=1018.060,280.748,-136.623,169.629,50.890,159.796
C04807=1018.054,280.500,-136.593,169.624,50.896,159.796
C04808=1018.048,280.252,-136.563,169.619,50.900,159.796
C04809=1018.042,280.003,-136.533,169.614,50.905,159.796
C04810=1018.035,279.756,-136.503,169.608,50.911,159.797
C04811=1018.029,279.508,-136.473,169.603,50.916,159.797
C04812=1018.024,279.260,-136.443,169.599,50.920,159.797
C04813=1018.018,279.028,-136.414,169.594,50.925,159.797
C04814=1018.012,278.796,-136.387,169.589,50.930,159.798
C04815=1018.006,278.563,-136.359,169.584,50.935,159.798
C04816=1018.001,278.332,-136.330,169.580,50.940,159.798
C04817=1017.996,278.100,-136.302,169.575,50.944,159.798
C04818=1017.989,277.868,-136.274,169.570,50.949,159.799
C04819=1017.984,277.637,-136.246,169.565,50.954,159.799
C04820=1017.978,277.405,-136.218,169.561,50.959,159.799
C04821=1017.973,277.156,-136.188,169.555,50.964,159.799
C04822=1017.966,276.909,-136.159,169.550,50.969,159.799
C04823=1017.960,276.660,-136.128,169.546,50.974,159.800
C04824=1017.955,276.412,-136.098,169.541,50.980,159.800
C04825=1017.948,276.164,-136.068,169.535,50.985,159.800
C04826=1017.942,275.916,-136.039,169.531,50.989,159.801
C04827=1017.936,275.668,-136.010,169.526,50.995,159.801
C04828=1017.930,275.420,-135.979,169.520,51.000,159.801
C04829=1017.924,275.171,-135.950,169.515,51.006,159.802
C04830=1017.918,274.923,-135.920,169.511,51.011,159.802
C04831=1017.911,274.675,-135.891,169.506,51.017,159.802
C04832=1017.906,274.427,-135.861,169.500,51.022,159.802
C04833=1017.899,274.179,-135.831,169.495,51.027,159.803
C04834=1017.894,273.931,-135.802,169.491,51.032,159.803
C04835=1017.888,273.682,-135.773,169.486,51.038,159.803
C04836=1017.882,273.435,-135.742,169.480,51.043,159.804
C04837=1017.876,273.187,-135.713,169.475,51.049,159.804
C04838=1017.869,272.937,-135.683,169.471,51.054,159.804
C04839=1017.863,272.689,-135.654,169.466,51.059,159.805
C04840=1017.857,272.441,-135.624,169.460,51.065,159.805
C04841=1017.851,272.193,-135.595,169.456,51.070,159.805
C04842=1017.846,271.945,-135.565,169.451,51.076,159.806
C04843=1017.839,271.697,-135.536,169.446,51.081,159.806
C04844=1017.833,271.449,-135.507,169.441,51.087,159.806
C04845=1017.827,271.201,-135.477,169.436,51.092,159.807
C04846=1017.821,270.953,-135.448,169.431,51.097,159.807
C04847=1017.816,270.704,-135.418,169.426,51.103,159.807
C04848=1017.809,270.456,-135.389,169.421,51.109,159.808
C04849=1017.803,270.208,-135.360,169.416,51.114,159.808
C04850=1017.798,269.959,-135.330,169.412,51.119,159.808
C04851=1017.791,269.711,-135.301,169.407,51.125,159.809
C04852=1017.786,269.463,-135.272,169.401,51.131,159.809
C04853=1017.780,269.215,-135.243,169.396,51.136,159.809
C04854=1017.773,268.967,-135.213,169.392,51.141,159.810
C04855=1017.767,268.719,-135.184,169.387,51.147,159.810
C04856=1017.762,268.471,-135.155,169.382,51.153,159.811
C04857=1017.756,268.223,-135.126,169.377,51.159,159.811
C04858=1017.750,267.975,-135.097,169.372,51.164,159.811
C04859=1017.743,267.726,-135.068,169.368,51.170,159.812
C04860=1017.738,267.478,-135.038,169.362,51.175,159.812
C04861=1017.732,267.229,-135.010,169.357,51.181,159.813
C04862=1017.726,266.981,-134.981,169.352,51.187,159.813
C04863=1017.719,266.733,-134.952,169.347,51.192,159.813
C04864=1017.714,266.484,-134.922,169.343,51.198,159.814
C04865=1017.708,266.236,-134.893,169.338,51.204,159.814
C04866=1017.701,265.988,-134.864,169.333,51.209,159.815
C04867=1017.696,265.740,-134.836,169.328,51.215,159.815
C04868=1017.690,265.492,-134.807,169.323,51.221,159.815
C04869=1017.684,265.244,-134.778,169.319,51.226,159.816
C04870=1017.678,264.995,-134.749,169.314,51.232,159.816
C04871=1017.672,264.747,-134.720,169.309,51.238,159.817
C04872=1017.666,264.499,-134.691,169.304,51.244,159.817
C04873=1017.660,264.270,-134.665,169.300,51.249,159.817
C04874=1017.655,264.039,-134.639,169.296,51.255,159.818
C04875=1017.649,263.810,-134.612,169.291,51.261,159.818
C04876=1017.644,263.580,-134.585,169.287,51.266,159.819
C04877=1017.638,263.351,-134.559,169.283,51.271,159.819
C04878=1017.632,263.121,-134.532,169.277,51.277,159.819
C04879=1017.627,262.891,-134.506,169.273,51.282,159.820
C04880=1017.622,262.662,-134.479,169.269,51.288,159.820
C04881=1017.616,262.413,-134.451,169.264,51.293,159.821
C04882=1017.610,262.165,-134.422,169.259,51.299,159.821
C04883=1017.604,261.917,-134.393,169.254,51.305,159.822
C04884=1017.598,261.668,-134.364,169.250,51.311,159.822
C04885=1017.593,261.420,-134.336,169.245,51.317,159.823
C04886=1017.586,261.172,-134.307,169.241,51.323,159.823
C04887=1017.580,260.923,-134.279,169.236,51.329,159.823
C04888=1017.575,260.676,-134.250,169.231,51.335,159.824
C04889=1017.569,260.427,-134.222,169.226,51.341,159.824
C04890=1017.563,260.179,-134.193,169.221,51.347,159.825
C04891=1017.557,259.930,-134.164,169.216,51.353,159.825
C04892=1017.551,259.682,-134.137,169.211,51.359,159.826
C04893=1017.545,259.434,-134.107,169.207,51.365,159.826
C04894=1017.538,259.186,-134.080,169.202,51.371,159.827
C04895=1017.533,258.938,-134.052,169.198,51.377,159.827
C04896=1017.527,258.689,-134.023,169.193,51.383,159.828
C04897=1017.520,258.441,-133.996,169.189,51.390,159.828
C04898=1017.514,258.192,-133.967,169.184,51.396,159.829
C04899=1017.509,257.944,-133.939,169.179,51.402,159.829
C04900=1017.502,257.696,-133.911,169.174,51.408,159.830
C04901=1017.496,257.447,-133.883,169.169,51.414,159.830
C04902=1017.490,257.199,-133.855,169.165,51.421,159.831
C04903=1017.484,256.951,-133.827,169.160,51.427,159.831
C04904=1017.478,256.702,-133.799,169.155,51.433,159.832
C04905=1017.472,256.454,-133.771,169.151,51.440,159.833
C04906=1017.466,256.205,-133.743,169.146,51.446,159.833
C04907=1017.460,255.957,-133.715,169.141,51.452,159.833
C04908=1017.454,255.709,-133.687,169.136,51.459,159.834
C04909=1017.448,255.460,-133.659,169.131,51.464,159.834
C04910=1017.443,255.212,-133.631,169.127,51.471,159.835
C04911=1017.436,254.964,-133.603,169.122,51.477,159.836
C04912=1017.430,254.715,-133.575,169.118,51.484,159.836
C04913=1017.424,254.467,-133.548,169.113,51.490,159.837
C04914=1017.418,254.218,-133.519,169.108,51.496,159.837
C04915=1017.413,253.970,-133.491,169.103,51.503,159.838
C04916=1017.406,253.722,-133.464,169.099,51.509,159.838
C04917=1017.400,253.473,-133.435,169.094,51.515,159.839
C04918=1017.395,253.225,-133.407,169.089,51.522,159.839
C04919=1017.388,252.977,-133.380,169.085,51.528,159.840
C04920=1017.383,252.728,-133.352,169.080,51.535,159.841
C04921=1017.377,252.480,-133.325,169.075,51.541,159.841
C04922=1017.371,252.232,-133.297,169.071,51.548,159.842
C04923=1017.365,251.983,-133.268,169.066,51.554,159.842
C04924=1017.359,251.735,-133.241,169.061,51.560,159.843
C04925=1017.353,251.486,-133.213,169.057,51.567,159.843
C04926=1017.348,251.238,-133.185,169.052,51.573,159.844
C04927=1017.342,250.989,-133.158,169.049,51.579,159.845
C04928=1017.336,250.741,-133.130,169.044,51.586,159.845
C04929=1017.330,250.492,-133.101,169.039,51.592,159.846
C04930=1017.324,250.245,-133.074,169.035,51.599,159.846
C04931=1017.319,249.996,-133.047,169.030,51.606,159.847
C04932=1017.312,249.748,-133.019,169.026,51.612,159.848
C04933=1017.307,249.517,-132.994,169.021,51.618,159.848
C04934=1017.302,249.287,-132.967,169.017,51.624,159.849
C04935=1017.297,249.056,-132.942,169.012,51.630,159.849
C04936=1017.291,248.825,-132.916,169.009,51.636,159.850
C04937=1017.286,248.595,-132.890,169.004,51.642,159.850
C04938=1017.281,248.364,-132.865,169.000,51.648,159.851
C04939=1017.276,248.135,-132.839,168.995,51.655,159.851
C04940=1017.270,247.904,-132.814,168.991,51.660,159.852
C04941=1017.264,247.655,-132.785,168.987,51.667,159.852
C04942=1017.258,247.407,-132.759,168.982,51.673,159.853
C04943=1017.253,247.159,-132.731,168.978,51.680,159.854
C04944=1017.246,246.910,-132.703,168.974,51.687,159.854
C04945=1017.241,246.661,-132.676,168.969,51.694,159.855
C04946=1017.236,246.413,-132.648,168.964,51.700,159.856
C04947=1017.230,246.164,-132.621,168.960,51.707,159.856
C04948=1017.224,245.916,-132.593,168.955,51.713,159.857
C04949=1017.218,245.669,-132.565,168.951,51.720,159.857
C04950=1017.213,245.419,-132.538,168.946,51.726,159.858
C04951=1017.207,245.171,-132.510,168.942,51.734,159.859
C04952=1017.201,244.923,-132.483,168.937,51.740,159.859
C04953=1017.196,244.675,-132.455,168.932,51.747,159.860
C04954=1017.190,244.425,-132.428,168.927,51.754,159.860
C04955=1017.184,244.178,-132.400,168.923,51.760,159.861
C04956=1017.179,243.929,-132.373,168.919,51.768,159.862
C04957=1017.174,243.681,-132.346,168.914,51.774,159.862
C04958=1017.168,243.432,-132.318,168.909,51.781,159.863
C04959=1017.163,243.183,-132.291,168.905,51.787,159.863
C04960=1017.156,242.935,-132.263,168.901,51.794,159.864
C04961=1017.151,242.687,-132.237,168.896,51.801,159.865
C04962=1017.145,242.438,-132.209,168.892,51.808,159.865
C04963=1017.139,242.190,-132.182,168.888,51.815,159.866
C04964=1017.133,241.942,-132.155,168.883,51.821,159.867
C04965=1017.128,241.693,-132.128,168.879,51.829,159.868
C04966=1017.122,241.444,-132.101,168.874,51.835,159.868
C04967=1017.116,241.196,-132.074,168.869,51.843,159.869
C04968=1017.111,240.947,-132.046,168.865,51.849,159.870
C04969=1017.105,240.699,-132.020,168.861,51.857,159.870
C04970=1017.099,240.451,-131.993,168.856,51.863,159.871
C04971=1017.093,240.201,-131.965,168.852,51.871,159.872
C04972=1017.088,239.953,-131.939,168.847,51.877,159.872
C04973=1017.082,239.705,-131.911,168.843,51.884,159.873
C04974=1017.077,239.457,-131.884,168.839,51.891,159.874
C04975=1017.071,239.208,-131.858,168.834,51.899,159.874
C04976=1017.064,238.959,-131.831,168.829,51.905,159.875
C04977=1017.059,238.711,-131.804,168.825,51.912,159.876
C04978=1017.053,238.462,-131.777,168.821,51.920,159.877
C04979=1017.047,238.214,-131.751,168.816,51.926,159.877
C04980=1017.041,237.966,-131.724,168.812,51.934,159.878
C04981=1017.036,237.717,-131.697,168.807,51.941,159.879
C04982=1017.031,237.469,-131.670,168.803,51.948,159.879
C04983=1017.025,237.220,-131.643,168.798,51.955,159.880
C04984=1017.018,236.971,-131.616,168.794,51.962,159.881
C04985=1017.013,236.723,-131.590,168.789,51.970,159.882
C04986=1017.007,236.475,-131.563,168.785,51.977,159.882
C04987=1017.001,236.226,-131.536,168.780,51.984,159.883
C04988=1016.996,235.977,-131.511,168.776,51.991,159.884
C04989=1016.990,235.729,-131.484,168.772,51.998,159.885
C04990=1016.984,235.481,-131.457,168.767,52.006,159.885
C04991=1016.978,235.232,-131.431,168.763,52.013,159.886
C04992=1016.973,234.984,-131.404,168.759,52.021,159.887
C04993=1016.967,234.750,-131.380,168.754,52.027,159.887
C04994=1016.961,234.516,-131.355,168.750,52.034,159.888
C04995=1016.956,234.282,-131.329,168.746,52.041,159.889
C04996=1016.951,234.049,-131.305,168.742,52.048,159.890
C04997=1016.945,233.815,-131.279,168.738,52.055,159.890
C04998=1016.940,233.580,-131.255,168.734,52.062,159.891
C04999=1016.934,233.347,-131.230,168.730,52.068,159.892
C05000=1016.929,233.113,-131.205,168.725,52.076,159.892
C05001=1016.923,232.864,-131.178,168.721,52.083,159.893
C05002=1016.918,232.615,-131.152,168.717,52.090,159.894
C05003=1016.912,232.367,-131.125,168.712,52.098,159.895
C05004=1016.906,232.119,-131.099,168.708,52.105,159.896
C05005=1016.901,231.870,-131.073,168.704,52.113,159.896
C05006=1016.895,231.621,-131.046,168.699,52.120,159.897
C05007=1016.889,231.372,-131.020,168.695,52.128,159.898
C05008=1016.884,231.124,-130.994,168.691,52.135,159.899
C05009=1016.878,230.876,-130.967,168.687,52.142,159.899
C05010=1016.873,230.627,-130.941,168.682,52.150,159.900
C05011=1016.867,230.379,-130.915,168.677,52.157,159.901
C05012=1016.861,230.131,-130.888,168.673,52.164,159.902
C05013=1016.856,229.882,-130.862,168.669,52.173,159.903
C05014=1016.849,229.634,-130.836,168.665,52.180,159.903
C05015=1016.844,229.385,-130.810,168.661,52.187,159.904
C05016=1016.838,229.136,-130.783,168.655,52.195,159.905
C05017=1016.833,228.887,-130.758,168.651,52.202,159.906
C05018=1016.827,228.639,-130.731,168.648,52.210,159.907
C05019=1016.821,228.390,-130.706,168.643,52.218,159.907
C05020=1016.815,228.141,-130.680,168.639,52.225,159.908
C05021=1016.810,227.894,-130.653,168.634,52.233,159.909
C05022=1016.805,227.645,-130.627,168.630,52.241,159.910
C05023=1016.799,227.396,-130.601,168.626,52.248,159.911
C05024=1016.793,227.147,-130.575,168.621,52.256,159.911
C05025=1016.787,226.899,-130.550,168.617,52.264,159.913
C05026=1016.781,226.650,-130.523,168.613,52.271,159.913
C05027=1016.776,226.401,-130.497,168.608,52.279,159.914
C05028=1016.770,226.153,-130.470,168.604,52.287,159.915
C05029=1016.764,225.905,-130.445,168.599,52.295,159.916
C05030=1016.759,225.656,-130.419,168.596,52.303,159.917
C05031=1016.753,225.407,-130.394,168.591,52.311,159.917
C05032=1016.747,225.158,-130.368,168.587,52.319,159.918
C05033=1016.741,224.910,-130.342,168.582,52.326,159.919
C05034=1016.735,224.661,-130.316,168.578,52.334,159.920
C05035=1016.730,224.413,-130.291,168.573,52.342,159.921
C05036=1016.724,224.164,-130.265,168.570,52.350,159.922
C05037=1016.719,223.915,-130.239,168.566,52.357,159.923
C05038=1016.713,223.667,-130.214,168.561,52.366,159.924
C05039=1016.707,223.418,-130.188,168.557,52.374,159.925
C05040=1016.701,223.170,-130.162,168.552,52.382,159.925
C05041=1016.696,222.921,-130.136,168.549,52.390,159.926
C05042=1016.690,222.673,-130.111,168.544,52.397,159.927
C05043=1016.684,222.424,-130.085,168.540,52.405,159.928
C05044=1016.679,222.175,-130.059,168.535,52.414,159.929
C05045=1016.673,221.927,-130.034,168.531,52.421,159.930
C05046=1016.668,221.678,-130.008,168.527,52.429,159.931
C05047=1016.661,221.429,-129.983,168.523,52.438,159.932
C05048=1016.656,221.180,-129.957,168.518,52.445,159.932
C05049=1016.650,220.932,-129.932,168.513,52.454,159.933
C05050=1016.645,220.683,-129.906,168.510,52.462,159.934
C05051=1016.639,220.435,-129.881,168.505,52.469,159.935
C05052=1016.633,220.186,-129.855,168.501,52.477,159.936
C05053=1016.628,219.948,-129.830,168.498,52.486,159.937
C05054=1016.622,219.710,-129.806,168.493,52.493,159.938
C05055=1016.617,219.473,-129.781,168.489,52.501,159.939
C05056=1016.612,219.234,-129.757,168.485,52.509,159.940
C05057=1016.607,218.996,-129.733,168.481,52.516,159.940
C05058=1016.601,218.758,-129.708,168.477,52.524,159.941
C05059=1016.596,218.521,-129.684,168.472,52.532,159.942
C05060=1016.591,218.282,-129.660,168.469,52.540,159.943
C05061=1016.585,218.033,-129.634,168.465,52.548,159.944
C05062=1016.580,217.785,-129.609,168.460,52.556,159.945
C05063=1016.574,217.536,-129.583,168.456,52.564,159.946
C05064=1016.568,217.288,-129.558,168.452,52.572,159.947
C05065=1016.562,217.039,-129.533,168.447,52.581,159.948
C05066=1016.556,216.790,-129.508,168.443,52.589,159.949
C05067=1016.551,216.542,-129.483,168.439,52.597,159.950
C05068=1016.545,216.293,-129.458,168.435,52.606,159.951
C05069=1016.539,216.044,-129.433,168.430,52.615,159.952
C05070=1016.534,215.796,-129.407,168.427,52.623,159.953
C05071=1016.528,215.547,-129.382,168.422,52.631,159.954
C05072=1016.523,215.298,-129.358,168.418,52.640,159.955
C05073=1016.516,215.050,-129.332,168.414,52.648,159.956
C05074=1016.511,214.801,-129.306,168.410,52.656,159.956
C05075=1016.506,214.552,-129.282,168.405,52.665,159.957
C05076=1016.499,214.304,-129.257,168.401,52.673,159.958
C05077=1016.494,214.056,-129.232,168.397,52.681,159.959
C05078=1016.489,213.806,-129.207,168.393,52.690,159.960
C05079=1016.483,213.558,-129.182,168.388,52.699,159.961
C05080=1016.477,213.309,-129.157,168.385,52.707,159.962
C05081=1016.471,213.060,-129.132,168.380,52.715,159.963
C05082=1016.466,212.812,-129.106,168.376,52.724,159.964
C05083=1016.460,212.562,-129.082,168.372,52.732,159.965
C05084=1016.454,212.314,-129.057,168.368,52.741,159.966
C05085=1016.449,212.065,-129.032,168.363,52.749,159.967
C05086=1016.444,211.817,-129.006,168.359,52.758,159.968
C05087=1016.438,211.568,-128.982,168.355,52.766,159.969
C05088=1016.432,211.320,-128.957,168.351,52.775,159.970
C05089=1016.426,211.070,-128.932,168.347,52.784,159.971
C05090=1016.421,210.822,-128.907,168.343,52.792,159.972
C05091=1016.416,210.573,-128.882,168.339,52.801,159.973
C05092=1016.410,210.325,-128.857,168.334,52.809,159.974
C05093=1016.404,210.076,-128.832,168.330,52.818,159.975
C05094=1016.398,209.828,-128.807,168.326,52.826,159.976
C05095=1016.393,209.578,-128.782,168.322,52.835,159.977
C05096=1016.388,209.330,-128.757,168.318,52.844,159.978
C05097=1016.382,209.081,-128.733,168.314,52.853,159.980
C05098=1016.376,208.832,-128.708,168.309,52.861,159.980
C05099=1016.371,208.584,-128.683,168.305,52.871,159.982
C05100=1016.365,208.335,-128.659,168.301,52.879,159.983
C05101=1016.360,208.086,-128.635,168.297,52.888,159.984
C05102=1016.354,207.837,-128.610,168.293,52.896,159.985
C05103=1016.348,207.589,-128.585,168.289,52.905,159.986
C05104=1016.342,207.340,-128.560,168.284,52.914,159.987
C05105=1016.337,207.091,-128.536,168.280,52.923,159.988
C05106=1016.332,206.843,-128.512,168.276,52.932,159.989
C05107=1016.325,206.594,-128.486,168.273,52.941,159.990
C05108=1016.320,206.345,-128.462,168.269,52.950,159.991
C05109=1016.315,206.097,-128.438,168.264,52.958,159.992
C05110=1016.309,205.847,-128.413,168.260,52.967,159.993
C05111=1016.304,205.599,-128.389,168.256,52.977,159.994
C05112=1016.297,205.350,-128.364,168.251,52.985,159.995
C05113=1016.292,205.112,-128.341,168.247,52.994,159.996
C05114=1016.287,204.874,-128.317,168.244,53.002,159.997
C05115=1016.282,204.637,-128.294,168.239,53.011,159.998
C05116=1016.276,204.399,-128.271,168.236,53.020,160.000
C05117=1016.271,204.161,-128.248,168.232,53.028,160.001
C05118=1016.266,203.923,-128.224,168.227,53.037,160.001
C05119=1016.260,203.684,-128.201,168.224,53.046,160.003
C05120=1016.254,203.447,-128.178,168.220,53.054,160.004
C05121=1016.236,202.432,-128.086,167.720,52.980,159.885
C05122=1016.231,202.182,-128.063,167.715,52.990,159.886
C05123=1016.226,201.934,-128.040,167.711,53.000,159.887
C05124=1016.222,201.685,-128.018,167.706,53.011,159.889
C05125=1016.217,201.437,-127.995,167.701,53.021,159.890
C05126=1016.213,201.187,-127.972,167.696,53.031,159.891
C05127=1016.208,200.938,-127.950,167.692,53.042,159.892
C05128=1016.203,200.689,-127.927,167.688,53.052,159.893
C05129=1016.199,200.440,-127.904,167.683,53.062,159.895
C05130=1016.194,200.192,-127.882,167.679,53.072,159.896
C05131=1016.189,199.942,-127.859,167.674,53.082,159.897
C05132=1016.185,199.693,-127.836,167.669,53.093,159.898
C05133=1016.180,199.445,-127.814,167.664,53.102,159.899
C05134=1016.176,199.196,-127.791,167.659,53.113,159.900
C05135=1016.171,198.947,-127.770,167.655,53.123,159.901
C05136=1016.167,198.697,-127.747,167.651,53.134,159.903
C05137=1016.162,198.448,-127.725,167.646,53.145,159.904
C05138=1016.157,198.199,-127.703,167.641,53.155,159.905
C05139=1016.153,197.951,-127.680,167.636,53.165,159.906
C05140=1016.148,197.702,-127.658,167.632,53.176,159.908
C05141=1016.142,197.453,-127.636,167.627,53.186,159.909
C05142=1016.138,197.204,-127.613,167.622,53.196,159.910
C05143=1016.133,196.955,-127.591,167.618,53.207,159.911
C05144=1016.129,196.706,-127.569,167.613,53.217,159.912
C05145=1016.124,196.457,-127.548,167.609,53.228,159.914
C05146=1016.120,196.208,-127.525,167.604,53.238,159.915
C05147=1016.115,195.959,-127.503,167.600,53.249,159.916
C05148=1016.110,195.710,-127.481,167.595,53.259,159.917
C05149=1016.105,195.460,-127.459,167.590,53.269,159.918
C05150=1016.101,195.212,-127.437,167.586,53.280,159.920
C05151=1016.096,194.963,-127.415,167.581,53.290,159.921
C05152=1016.092,194.714,-127.392,167.577,53.300,159.922
C05153=1016.087,194.465,-127.371,167.573,53.311,159.923
C05154=1016.082,194.216,-127.349,167.569,53.322,159.925
C05155=1016.077,193.967,-127.327,167.564,53.332,159.926
C05156=1016.073,193.718,-127.304,167.559,53.342,159.927
C05157=1016.068,193.469,-127.283,167.555,53.353,159.928
C05158=1016.064,193.220,-127.261,167.550,53.363,159.929
C05159=1016.060,192.971,-127.239,167.545,53.374,159.930
C05160=1016.055,192.722,-127.217,167.541,53.384,159.932
C05161=1016.050,192.473,-127.195,167.536,53.394,159.933
C05162=1016.045,192.224,-127.173,167.533,53.404,159.934
C05163=1016.041,191.975,-127.151,167.528,53.416,159.936
C05164=1016.036,191.726,-127.129,167.524,53.426,159.937
C05165=1016.031,191.478,-127.107,167.519,53.436,159.938
C05166=1016.027,191.228,-127.086,167.515,53.447,159.939
C05167=1016.023,190.979,-127.064,167.510,53.457,159.940
C05168=1016.018,190.730,-127.042,167.505,53.468,159.941
C05169=1016.013,190.481,-127.020,167.502,53.478,159.943
C05170=1016.009,190.232,-126.997,167.497,53.488,159.944
C05171=1016.005,189.983,-126.976,167.493,53.498,159.945
C05172=1016.000,189.734,-126.954,167.489,53.510,159.946
C05173=1015.995,189.485,-126.932,167.484,53.520,159.948
C05174=1015.991,189.236,-126.910,167.479,53.530,159.949
C05175=1015.986,188.987,-126.889,167.476,53.540,159.950
C05176=1015.982,188.738,-126.867,167.471,53.551,159.951
C05177=1015.977,188.489,-126.845,167.467,53.561,159.952
C05178=1015.973,188.241,-126.823,167.462,53.572,159.954
C05179=1015.969,187.991,-126.802,167.457,53.582,159.955
C05180=1015.964,187.742,-126.780,167.454,53.592,159.956
C05181=1015.960,187.493,-126.758,167.449,53.603,159.957
C05182=1015.955,187.213,-126.734,167.445,53.615,159.959
C05183=1015.949,186.933,-126.709,167.440,53.626,159.960
C05184=1015.944,186.653,-126.685,167.435,53.639,159.962
C05185=1015.940,186.373,-126.660,167.431,53.650,159.963
C05186=1015.935,186.124,-126.638,167.426,53.660,159.964
C05187=1015.931,185.875,-126.617,167.422,53.671,159.965
C05188=1015.926,185.626,-126.595,167.417,53.681,159.967
C05189=1015.922,185.378,-126.573,167.414,53.691,159.968
C05190=1015.918,185.128,-126.552,167.409,53.702,159.969
C05191=1015.913,184.879,-126.530,167.404,53.712,159.970
C05192=1015.908,184.630,-126.509,167.401,53.722,159.972
C05193=1015.904,184.381,-126.486,167.397,53.733,159.973
C05194=1015.900,184.132,-126.466,167.392,53.744,159.974
C05195=1015.896,183.883,-126.444,167.388,53.754,159.975
C05196=1015.891,183.634,-126.421,167.384,53.764,159.977
C05197=1015.887,183.385,-126.400,167.380,53.775,159.978
C05198=1015.883,183.136,-126.379,167.375,53.785,159.979
C05199=1015.878,182.887,-126.358,167.372,53.795,159.980
C05200=1015.874,182.638,-126.335,167.367,53.806,159.981
C05201=1015.870,182.388,-126.314,167.363,53.816,159.983
C05202=1015.865,182.140,-126.292,167.359,53.827,159.984
C05203=1015.861,181.891,-126.271,167.355,53.837,159.985
C05204=1015.857,181.641,-126.250,167.350,53.848,159.986
C05205=1015.852,181.392,-126.229,167.347,53.858,159.988
C05206=1015.847,181.143,-126.207,167.343,53.869,159.989
C05207=1015.842,180.894,-126.186,167.339,53.880,159.991
C05208=1015.838,180.645,-126.166,167.334,53.891,159.992
C05209=1015.833,180.396,-126.145,167.330,53.902,159.993
C05210=1015.828,180.147,-126.124,167.326,53.912,159.994
C05211=1015.824,179.897,-126.103,167.321,53.923,159.995
C05212=1015.820,179.649,-126.082,167.318,53.934,159.997
C05213=1015.814,179.400,-126.062,167.314,53.944,159.998
C05214=1015.810,179.150,-126.040,167.310,53.955,160.000
C05215=1015.805,178.901,-126.020,167.305,53.966,160.001
C05216=1015.800,178.653,-125.998,167.301,53.976,160.002
C05217=1015.796,178.403,-125.977,167.298,53.987,160.004
C05218=1015.791,178.154,-125.957,167.293,53.998,160.005
C05219=1015.787,177.906,-125.936,167.289,54.009,160.006
C05220=1015.782,177.656,-125.915,167.285,54.019,160.007
C05221=1015.777,177.407,-125.894,167.280,54.030,160.009
C05222=1015.772,177.158,-125.873,167.277,54.041,160.010
C05223=1015.768,176.909,-125.853,167.273,54.051,160.011
C05224=1015.763,176.660,-125.832,167.268,54.062,160.012
C05225=1015.759,176.410,-125.811,167.264,54.073,160.014
C05226=1015.754,176.162,-125.790,167.260,54.084,160.015
C05227=1015.750,175.912,-125.770,167.257,54.095,160.017
C05228=1015.745,175.663,-125.750,167.252,54.105,160.018
C05229=1015.741,175.414,-125.729,167.248,54.116,160.019
C05230=1015.736,175.165,-125.707,167.244,54.127,160.020
C05231=1015.731,174.916,-125.687,167.241,54.137,160.022
C05232=1015.727,174.667,-125.666,167.236,54.148,160.023
C05233=1015.722,174.418,-125.646,167.232,54.159,160.024
C05234=1015.718,174.169,-125.625,167.229,54.169,160.026
C05235=1015.713,173.919,-125.604,167.225,54.180,160.027
C05236=1015.709,173.671,-125.583,167.220,54.191,160.028
C05237=1015.704,173.422,-125.562,167.216,54.201,160.029
C05238=1015.699,173.172,-125.542,167.213,54.212,160.031
C05239=1015.695,172.923,-125.522,167.209,54.223,160.032
C05240=1015.691,172.674,-125.501,167.204,54.233,160.033
C05241=1015.686,172.425,-125.480,167.201,54.244,160.035
C05242=1015.682,172.176,-125.459,167.197,54.255,160.036
C05243=1015.677,171.927,-125.439,167.192,54.266,160.037
C05244=1015.673,171.677,-125.419,167.190,54.276,160.039
C05245=1015.668,171.428,-125.397,167.185,54.287,160.040
C05246=1015.662,171.073,-125.368,167.180,54.302,160.042
C05247=1015.656,170.717,-125.339,167.174,54.318,160.044
C05248=1015.649,170.362,-125.309,167.168,54.333,160.046
C05249=1015.643,170.006,-125.280,167.163,54.348,160.048
C05250=1015.638,169.757,-125.260,167.159,54.358,160.049
C05251=1015.634,169.508,-125.239,167.155,54.370,160.050
C05252=1015.629,169.259,-125.219,167.152,54.380,160.052
C05253=1015.625,169.010,-125.198,167.147,54.391,160.053
C05254=1015.621,168.760,-125.177,167.144,54.402,160.054
C05255=1015.616,168.512,-125.157,167.140,54.412,160.056
C05256=1015.612,168.263,-125.137,167.136,54.423,160.057
C05257=1015.607,168.013,-125.117,167.133,54.434,160.058
C05258=1015.603,167.764,-125.096,167.128,54.444,160.060
C05259=1015.599,167.515,-125.075,167.125,54.454,160.061
C05260=1015.594,167.266,-125.055,167.121,54.466,160.062
C05261=1015.590,167.016,-125.034,167.117,54.476,160.064
C05262=1015.585,166.768,-125.014,167.113,54.487,160.065
C05263=1015.581,166.518,-124.994,167.109,54.497,160.066
C05264=1015.577,166.269,-124.973,167.106,54.508,160.068
C05265=1015.572,166.021,-124.953,167.102,54.519,160.069
C05266=1015.568,165.771,-124.932,167.099,54.529,160.070
C05267=1015.563,165.522,-124.912,167.095,54.540,160.072
C05268=1015.559,165.272,-124.891,167.091,54.551,160.073
C05269=1015.555,165.024,-124.871,167.087,54.561,160.074
C05270=1015.551,164.775,-124.851,167.084,54.572,160.075
C05271=1015.546,164.525,-124.830,167.080,54.583,160.077
C05272=1015.542,164.277,-124.810,167.077,54.593,160.078
C05273=1015.538,164.027,-124.789,167.072,54.604,160.079
C05274=1015.533,163.778,-124.769,167.069,54.614,160.081
C05275=1015.529,163.529,-124.749,167.065,54.625,160.082
C05276=1015.525,163.279,-124.728,167.062,54.636,160.084
C05277=1015.520,163.031,-124.708,167.057,54.646,160.085
C05278=1015.517,162.782,-124.688,167.054,54.657,160.086
C05279=1015.511,162.533,-124.667,167.050,54.668,160.088
C05280=1015.508,162.283,-124.647,167.047,54.678,160.089
C05281=1015.503,162.035,-124.627,167.043,54.689,160.090
C05282=1015.499,161.785,-124.607,167.039,54.699,160.091
C05283=1015.495,161.536,-124.586,167.036,54.711,160.093
C05284=1015.491,161.287,-124.566,167.032,54.721,160.094
C05285=1015.486,161.037,-124.545,167.028,54.731,160.095
C05286=1015.483,160.826,-124.529,167.025,54.741,160.097
C05287=1015.479,160.615,-124.512,167.022,54.749,160.098
C05288=1015.476,160.404,-124.494,167.019,54.758,160.099
C05289=1015.472,160.192,-124.478,167.017,54.767,160.100
C05290=1015.468,159.981,-124.460,167.013,54.776,160.101
C05291=1015.465,159.769,-124.443,167.010,54.785,160.102
C05292=1015.461,159.558,-124.425,167.007,54.795,160.103
C05293=1015.457,159.346,-124.409,167.004,54.803,160.104
C05294=1015.454,159.097,-124.388,167.000,54.813,160.106
C05295=1015.449,158.847,-124.368,166.997,54.825,160.107
C05296=1015.445,158.598,-124.348,166.993,54.835,160.109
C05297=1015.441,158.349,-124.327,166.990,54.845,160.110
C05298=1015.436,158.100,-124.308,166.986,54.856,160.111
C05299=1015.432,157.851,-124.288,166.982,54.868,160.113
C05300=1015.427,157.602,-124.269,166.979,54.878,160.114
C05301=1015.422,157.352,-124.249,166.975,54.889,160.115
C05302=1015.418,157.103,-124.229,166.972,54.900,160.117
C05303=1015.414,156.854,-124.210,166.968,54.911,160.118
C05304=1015.409,156.605,-124.190,166.965,54.921,160.120
C05305=1015.405,156.355,-124.169,166.961,54.932,160.121
C05306=1015.401,156.106,-124.150,166.958,54.943,160.122
C05307=1015.396,155.857,-124.130,166.954,54.954,160.124
C05308=1015.392,155.608,-124.111,166.951,54.965,160.125
C05309=1015.387,155.359,-124.091,166.947,54.975,160.126
C05310=1015.382,155.078,-124.069,166.944,54.988,160.128
C05311=1015.377,154.798,-124.047,166.939,54.999,160.129
C05312=1015.372,154.517,-124.025,166.936,55.012,160.131
C05313=1015.368,154.237,-124.003,166.931,55.024,160.133
C05314=1015.363,153.988,-123.984,166.927,55.035,160.134
C05315=1015.358,153.738,-123.964,166.924,55.046,160.135
C05316=1015.354,153.489,-123.944,166.921,55.056,160.137
C05317=1015.350,153.240,-123.925,166.917,55.067,160.138
C05318=1015.346,152.991,-123.905,166.914,55.078,160.140
C05319=1015.342,152.742,-123.885,166.910,55.089,160.141
C05320=1015.337,152.492,-123.866,166.907,55.099,160.142
C05321=1015.332,152.243,-123.846,166.903,55.111,160.144
C05322=1015.328,151.994,-123.827,166.900,55.121,160.145
C05323=1015.324,151.745,-123.807,166.896,55.132,160.146
C05324=1015.319,151.496,-123.788,166.893,55.143,160.148
C05325=1015.314,151.247,-123.769,166.889,55.154,160.149
C05326=1015.310,150.998,-123.749,166.886,55.165,160.151
C05327=1015.305,150.748,-123.730,166.882,55.175,160.152
C05328=1015.301,150.499,-123.711,166.879,55.186,160.153
C05329=1015.296,150.250,-123.691,166.875,55.197,160.155
C05330=1015.292,150.001,-123.672,166.873,55.208,160.156
C05331=1015.288,149.751,-123.652,166.868,55.219,160.157
C05332=1015.283,149.502,-123.633,166.865,55.229,160.159
C05333=1015.279,149.253,-123.614,166.863,55.240,160.160
C05334=1015.275,149.004,-123.595,166.858,55.251,160.162
C05335=1015.270,148.754,-123.575,166.856,55.262,160.163
C05336=1015.266,148.505,-123.555,166.852,55.273,160.165
C05337=1015.261,148.256,-123.536,166.848,55.283,160.166
C05338=1015.257,148.006,-123.517,166.845,55.295,160.167
C05339=1015.253,147.757,-123.498,166.842,55.305,160.169
C05340=1015.248,147.508,-123.479,166.839,55.316,160.170
C05341=1015.244,147.259,-123.459,166.835,55.327,160.172
C05342=1015.240,147.010,-123.440,166.832,55.338,160.173
C05343=1015.235,146.761,-123.421,166.828,55.349,160.174
C05344=1015.231,146.512,-123.402,166.825,55.359,160.176
C05345=1015.227,146.262,-123.383,166.822,55.370,160.177
C05346=1015.222,146.013,-123.363,166.818,55.381,160.179
C05347=1015.217,145.764,-123.344,166.815,55.392,160.180
C05348=1015.213,145.515,-123.326,166.811,55.403,160.181
C05349=1015.209,145.266,-123.306,166.808,55.414,160.183
C05350=1015.205,145.016,-123.287,166.805,55.424,160.184
C05351=1015.200,144.767,-123.269,166.802,55.436,160.186
C05352=1015.195,144.517,-123.249,166.799,55.446,160.187
C05353=1015.191,144.268,-123.230,166.795,55.458,160.189
C05354=1015.186,144.019,-123.211,166.792,55.468,160.190
C05355=1015.182,143.769,-123.192,166.788,55.479,160.191
C05356=1015.177,143.520,-123.173,166.785,55.490,160.193
C05357=1015.173,143.271,-123.155,166.781,55.501,160.194
C05358=1015.168,143.022,-123.135,166.779,55.512,160.196
C05359=1015.164,142.772,-123.116,166.776,55.522,160.197
C05360=1015.159,142.524,-123.098,166.772,55.534,160.198
C05361=1015.155,142.274,-123.079,166.769,55.544,160.200
C05362=1015.151,142.025,-123.059,166.765,55.555,160.201
C05363=1015.146,141.775,-123.041,166.762,55.566,160.203
